(* PLC project measure36, PHOENIX CONTACT Software MULTIPROG 5.51 *)
(* stored: companyURL https://www.phoenixcontact-software.com, productRelease Build 473, creationDateTime 2024-06-25T14:51:15, contentDescription ###XMLINFO=2;1;2;;, version 0.1.75, modificationDateTime 2024-06-25T14:51:15 *)

PROGRAM mainST
  VAR
    input01 : BOOL;  (* 入力01 *)
    resLD : BOOL;
    resLDB : BOOL;
    C005 : BOOL;
    resAND : BOOL;
    C007 : BOOL;
    resANB : BOOL;
    C010 : BOOL;
    resOR : BOOL;
    C015 : BOOL;
    resORB : BOOL;
    resOUT : BOOL;
    resOUB : BOOL;
    resSET : BOOL;
    C024 : BOOL;
    resRES : BOOL;
    inTIMER01 : BOOL;
    TON_1 : TON;
    passed01 : TIME;
    TON_2 : TON;
    passed02 : TIME;
    resLD_T01 : BOOL;
    resLD_T02 : BOOL;
    inCounter : BOOL;
    enableCnt : BOOL;
    CTU_1 : CTU;
    outConter : BOOL;
    valCounter : INT;
    inTimER02 : BOOL;
    TON_3 : TON;
    passed03 : TIME;
    resT5 : BOOL;
    resLDB_T : BOOL;
    inCounter2 : BOOL;
    CTU_2 : CTU;
    outConter2 : BOOL;
    valCounter2 : INT;
    resLDB_C : BOOL;
    resLD_C : BOOL;
    inTimeR03 : BOOL;
    TON_4 : TON;
    outTimer : BOOL;
    passed04 : TIME;
    C046 : BOOL;
    resAND_T : BOOL;
    resTimer01 : BOOL;
    resTimer02 : BOOL;
    inCounter3 : BOOL;
    CTU_3 : CTU;
    outCounter3 : BOOL;
    valCounter3 : INT;
    C052 : BOOL;
    resAND_C : BOOL;
    inTimer05 : BOOL;
    TON_5 : TON;
    outTimer05 : BOOL;
    passed05 : TIME;
    C055 : BOOL;
    resANB_T : BOOL;
    inCounter04 : BOOL;
    CTU_4 : CTU;
    valCounter04 : INT;
    outConter04 : BOOL;
    C061 : BOOL;
    resANB_C : BOOL;
    inTimer06 : BOOL;
    TON_6 : TON;
    outTimer06 : BOOL;
    passed06 : TIME;
    resOR_T : BOOL;
    inCounter05 : BOOL;
    CTU_5 : CTU;
    outCounter05 : BOOL;
    valCounter05 : INT;
    resOR_C : BOOL;
    inTimer07 : BOOL;
    TON_7 : TON;
    outTimer07 : BOOL;
    passed07 : TIME;
    resORB_T : BOOL;
    inCounter06 : BOOL;
    CTU_6 : CTU;
    outCounter06 : BOOL;
    valCounter06 : INT;
    resORB_C : BOOL;
    C083 : BOOL;
    C085 : BOOL;
    resANL : BOOL;
    C089 : BOOL;
    C091 : BOOL;
    resORL : BOOL;
    setten0101 : BOOL;
    setten0102 : BOOL;
    setten0103 : BOOL;
    setten0104 : BOOL;
    resCoil01 : BOOL;
    setten0204 : BOOL;
    setten0304 : BOOL;
    resCoil02 : BOOL;
    resCoil03 : BOOL;
    setten0403 : BOOL;
    setten0503 : BOOL;
    resCoil04 : BOOL;
    resCoil05 : BOOL;
    setten0603 : BOOL;
    setten0702 : BOOL;
    setten0802 : BOOL;
    setten0902 : BOOL;
    resCoil07 : BOOL;
    resCoil06 : BOOL;
    resCoil08 : BOOL;
    resCoil09 : BOOL;
    C065 : BOOL;
    C069 : BOOL;
    C075 : BOOL;
    C078 : BOOL;
    inBia0101 : BOOL;
    inBia0102 : BOOL;
    inBia0202 : BOOL;
    inBia0203 : BOOL;
    inBia0303 : BOOL;
    inBIa0404 : BOOL;
    inBIa0504 : BOOL;
    resBia01 : BOOL;
    resBia02 : BOOL;
    resBia03 : BOOL;
    inCLR01 : BOOL;
    resCLR01 : BOOL;
    inCLR02 : BOOL;
    resCLR02 : BOOL;
    inCLR03 : BOOL;
    resCLR03 : BOOL;
    inCLR0401 : BOOL;
    inCLR0402 : BOOL;
    resCLR04 : BOOL;
    F_TRIG_1 : F_TRIG;
    inDIFU : BOOL;
    outDIFU : BOOL;
    resDIFU : BOOL;
    holdDIFU : BOOL;
    inDIFD : BOOL;
    R_TRIG_1 : R_TRIG;
    outDIFD : BOOL;
    holdDIFD : BOOL;
    resDIFD : BOOL;
    TotalCount : UINT;
    switch : BOOL;
  END_VAR
  VAR_EXTERNAL
    ECAT_Slave1_DI1 : BOOL;
  END_VAR
  VAR
    CTU_7 : CTU;
  END_VAR
  VAR_EXTERNAL
    ECAT_Slave4_AO1 : INT;
  END_VAR
  VAR
    CT_Reset : BOOL;
  END_VAR
  VAR_EXTERNAL
    ECAT_Slave5_DI1 : BOOL;
    ECAT_Slave5_DO1 : BOOL;
  END_VAR
  VAR
    IL変数_1 : BOOL;
    IL変数_2 : BOOL;
    IL変数_3 : BOOL;
    IL変数_4 : BOOL;
    IL変数_5 : BOOL;
    IL変数_6 : BOOL;
    IL変数_7 : BOOL;
    IL変数_8 : BOOL;
    IL変数_9 : BOOL;
    IL変数_10 : BOOL;
    IL変数_11 : BOOL;
    IL変数_12 : BOOL;
    IL変数_13 : BOOL;
    IL変数_14 : BOOL;
    IL変数_15 : BOOL;
    IL変数_16 : BOOL;
    IL変数_17 : BOOL;
    IL変数_18 : BOOL;
    IL変数_19 : BOOL;
    IL変数_20 : BOOL;
    IL変数_21 : BOOL;
    IL変数_22 : BOOL;
    IL変数_23 : BOOL;
    IL変数_24 : BOOL;
    IL変数_25 : BOOL;
    IL変数_26 : BOOL;
    IL変数_27 : BOOL;
    IL変数_28 : BOOL;
    IL変数_29 : BOOL;
    IL変数_30 : BOOL;
    IL変数_31 : BOOL;
    IL変数_32 : BOOL;
    IL変数_33 : BOOL;
    IL変数_34 : BOOL;
    IL変数_35 : BOOL;
    IL変数_36 : BOOL;
    IL変数_37 : BOOL;
    IL変数_38 : BOOL;
    IL変数_39 : BOOL;
    IL変数_40 : BOOL;
    IL変数_41 : BOOL;
    IL変数_42 : BOOL;
    IL変数_43 : BOOL;
    IL変数_44 : BOOL;
    IL変数_45 : BOOL;
    IL変数_46 : BOOL;
    IL変数_47 : BOOL;
    IL変数_48 : BOOL;
    IL変数_49 : BOOL;
    IL変数_50 : BOOL;
    IL変数_51 : BOOL;
    IL変数_52 : BOOL;
    IL変数_53 : BOOL;
    IL変数_54 : BOOL;
    IL変数_55 : BOOL;
    IL変数_56 : BOOL;
    IL変数_57 : BOOL;
    IL変数_58 : BOOL;
    IL変数_59 : BOOL;
    IL変数_60 : BOOL;
    IL変数_61 : BOOL;
    IL変数_62 : BOOL;
    IL変数_63 : BOOL;
    IL変数_64 : BOOL;
    IL変数_65 : BOOL;
    IL変数_66 : BOOL;
    IL変数_67 : BOOL;
    IL変数_68 : BOOL;
    IL変数_69 : BOOL;
    IL変数_70 : BOOL;
    IL変数_71 : BOOL;
    IL変数_72 : BOOL;
    IL変数_73 : BOOL;
    IL変数_74 : BOOL;
    IL変数_75 : BOOL;
    IL変数_76 : BOOL;
    IL変数_77 : BOOL;
    IL変数_78 : BOOL;
    IL変数_79 : BOOL;
    IL変数_80 : BOOL;
    IL変数_81 : BOOL;
    IL変数_82 : BOOL;
    IL変数_83 : BOOL;
    IL変数_84 : BOOL;
    IL変数_85 : BOOL;
    IL変数_86 : BOOL;
    IL変数_87 : BOOL;
    IL変数_88 : BOOL;
    IL変数_89 : BOOL;
    IL変数_90 : BOOL;
    IL変数_91 : BOOL;
    IL変数_92 : BOOL;
    IL変数_93 : BOOL;
    IL変数_94 : BOOL;
    IL変数_95 : BOOL;
    IL変数_96 : BOOL;
    IL変数_97 : BOOL;
    IL変数_98 : BOOL;
    IL変数_99 : BOOL;
    IL変数_100 : BOOL;
    IL変数_101 : BOOL;
    IL変数_102 : BOOL;
    IL変数_103 : BOOL;
    IL変数_104 : BOOL;
    IL変数_105 : BOOL;
    IL変数_106 : BOOL;
    IL変数_107 : BOOL;
    IL変数_108 : BOOL;
    IL変数_109 : BOOL;
    IL変数_110 : BOOL;
    IL変数_111 : BOOL;
    IL変数_112 : BOOL;
    IL変数_113 : BOOL;
    IL変数_114 : BOOL;
    IL変数_115 : BOOL;
    IL変数_116 : BOOL;
    IL変数_117 : BOOL;
    IL変数_118 : BOOL;
    IL変数_119 : BOOL;
    IL変数_120 : BOOL;
    IL変数_121 : BOOL;
    IL変数_122 : BOOL;
    IL変数_123 : BOOL;
    IL変数_124 : BOOL;
    IL変数_125 : BOOL;
    IL変数_126 : BOOL;
    IL変数_127 : BOOL;
    IL変数_128 : BOOL;
    IL変数_129 : BOOL;
    IL変数_130 : BOOL;
    IL変数_131 : BOOL;
    IL変数_132 : BOOL;
    IL変数_133 : BOOL;
    IL変数_134 : BOOL;
    IL変数_135 : BOOL;
    IL変数_136 : BOOL;
    IL変数_137 : BOOL;
    IL変数_138 : BOOL;
    IL変数_139 : BOOL;
    IL変数_140 : BOOL;
    IL変数_141 : BOOL;
    IL変数_142 : BOOL;
    IL変数_143 : BOOL;
    IL変数_144 : BOOL;
    IL変数_145 : BOOL;
    IL変数_146 : BOOL;
    IL変数_147 : BOOL;
    IL変数_148 : BOOL;
    IL変数_149 : BOOL;
    IL変数_150 : BOOL;
    IL変数_151 : BOOL;
    IL変数_152 : BOOL;
    IL変数_153 : BOOL;
    IL変数_154 : BOOL;
    IL変数_155 : BOOL;
    IL変数_156 : BOOL;
    IL変数_157 : BOOL;
    IL変数_158 : BOOL;
    IL変数_159 : BOOL;
    IL変数_160 : BOOL;
    IL変数_161 : BOOL;
    IL変数_162 : BOOL;
    IL変数_163 : BOOL;
    IL変数_164 : BOOL;
    IL変数_165 : BOOL;
    IL変数_166 : BOOL;
    IL変数_167 : BOOL;
    IL変数_168 : BOOL;
    IL変数_169 : BOOL;
    IL変数_170 : BOOL;
    IL変数_171 : BOOL;
    IL変数_172 : BOOL;
    IL変数_173 : BOOL;
    IL変数_174 : BOOL;
    IL変数_175 : BOOL;
    IL変数_176 : BOOL;
    IL変数_177 : BOOL;
    IL変数_178 : BOOL;
    IL変数_179 : BOOL;
    IL変数_180 : BOOL;
  END_VAR

						
							
								
							
							
								(**** 全命令テスト ****)
(**** 回路ON ****)
LD		ECAT_Slave5_DI1
ST		input01
ST		inBia0101
ST		inBia0102
ST		inBia0202
ST		inBia0203
ST		inBia0303
ST		inBIa0404
ST		inBIa0504
ST		inCLR01
ST		inCLR02
ST		inCLR03
ST		inCLR0401
ST		inCLR0402
ST		inCounter
ST		inCounter2
ST		inCounter3
ST		inCounter04
ST		inCounter05
ST		inCounter06
ST		inDIFU
ST		inDIFD
ST		inTIMER01
ST		inTimER02
ST		inTimeR03
ST		inTimer05
ST		inTimer06
ST		inTimer07
									
								
							
						
					
						
							
								
							
							
								(*■LD命令*)
LD		input01
ST		resLD
									
(*■LDB命令*)
LDN		input01
STN		resLDB
									
(*■AND命令*)
LDN		C005
AND		input01
ST		resAND
									
(*■ANB命令*)
LDN		C007
ANDN		input01
STN		resANB
									
(*■OR命令*)
LD		C010
OR		input01
ST		resOR
									
(*■ORB命令*)
LD		C015
ORN		input01
STN		resORB
									
(*■OUT命令*)
LD		input01
ST		resOUT
									
(*■OUB命令*)
LDN		input01
STN		resOUB
									
(*■SET命令*)
LD		input01
ANDN		resSET
S		resSET
									
(*■RES命令*)
LD		input01
S		C024
									
LD		input01
R		C024
									
LDN		C024
ST		resRES
									
(*■LD_T命令*)
LD		inTIMER01
ST		TON_1.IN
ST		TON_2.IN
LD		TIME#30s
ST		TON_1.PT
CAL		TON_1
LD		TON_1.Q
ST		resTimer01
LD		TON_1.ET
ST		passed01
LD		TIME#1m
ST		TON_2.PT
CAL		TON_2
LD		TON_2.Q
ST		resTimer02
LD		TON_2.ET
ST		passed02
									
LD		resTimer01
ST		resLD_T01
									
LD		resTimer02
ST		resLD_T02
									
(*■LD_C命令*)
LD		inCounter
ST		CTU_1.CU
LD		enableCnt
ST		CTU_1.RESET
LD		INT#5000
ST		CTU_1.PV
CAL		CTU_1
LD		CTU_1.Q
ST		outConter
LD		CTU_1.CV
ST		valCounter
									
LD		outConter
ST		resLD_C
									
(*■LDB_T命令*)
LD		inTimER02
ST		TON_3.IN
LD		TIME#30s
ST		TON_3.PT
CAL		TON_3
LD		TON_3.Q
ST		resT5
LD		TON_3.ET
ST		passed03
									
LDN		resT5
STN		resLDB_T
									
(*■LDB_C命令*)
LD		inCounter2
ST		CTU_2.CU
LD		enableCnt
ST		CTU_2.RESET
LD		INT#5000
ST		CTU_2.PV
CAL		CTU_2
LD		CTU_2.Q
ST		outConter2
LD		CTU_2.CV
ST		valCounter2
									
LDN		outConter2
STN		resLDB_C
									
(*■AND_T命令*)
LD		inTimeR03
ST		TON_4.IN
LD		TIME#30s
ST		TON_4.PT
CAL		TON_4
LD		TON_4.Q
ST		outTimer
LD		TON_4.ET
ST		passed04
									
LDN		C046
AND		outTimer
ST		resAND_T
									
(*■AND_C命令*)
LD		inCounter3
ST		CTU_3.CU
LD		enableCnt
ST		CTU_3.RESET
LD		INT#5000
ST		CTU_3.PV
CAL		CTU_3
LD		CTU_3.Q
ST		outCounter3
LD		CTU_3.CV
ST		valCounter3
									
LDN		C052
AND		outCounter3
ST		resAND_C
									
(*■ANB_T命令*)
LD		inTimer05
ST		TON_5.IN
LD		TIME#30s
ST		TON_5.PT
CAL		TON_5
LD		TON_5.Q
ST		outTimer05
LD		TON_5.ET
ST		passed05
									
LDN		C055
ANDN		outTimer05
STN		resANB_T
									
(*■ANB_C命令*)
LD		inCounter04
ST		CTU_4.CU
LD		enableCnt
ST		CTU_4.RESET
LD		INT#5000
ST		CTU_4.PV
CAL		CTU_4
LD		CTU_4.Q
ST		outConter04
LD		CTU_4.CV
ST		valCounter04
									
LDN		C061
ANDN		outConter04
STN		resANB_C
									
(*■OR_T命令*)
LD		inTimer06
ST		TON_6.IN
LD		TIME#30s
ST		TON_6.PT
CAL		TON_6
LD		TON_6.Q
ST		outTimer06
LD		TON_6.ET
ST		passed06
									
LD		C065
OR		outTimer06
ST		resOR_T
									
(*■OR_C命令*)
LD		inCounter05
ST		CTU_5.CU
LD		enableCnt
ST		CTU_5.RESET
LD		INT#5000
ST		CTU_5.PV
CAL		CTU_5
LD		CTU_5.Q
ST		outCounter05
LD		CTU_5.CV
ST		valCounter05
									
LD		C069
OR		outCounter05
ST		resOR_C
									
(*■ORB_T命令*)
LD		inTimer07
ST		TON_7.IN
LD		TIME#30s
ST		TON_7.PT
CAL		TON_7
LD		TON_7.Q
ST		outTimer07
LD		TON_7.ET
ST		passed07
									
LD		C075
ORN		outTimer07
STN		resORB_T
									
(*■ORB_C命令*)
LD		inCounter06
ST		CTU_6.CU
LD		enableCnt
ST		CTU_6.RESET
LD		INT#5000
ST		CTU_6.PV
CAL		CTU_6
LD		CTU_6.Q
ST		outCounter06
LD		CTU_6.CV
ST		valCounter06
									
LD		C078
ORN		outCounter06
STN		resORB_C
									
(*■ANL命令*)
LD		input01
OR		C083
ST		IL変数_1
LD		input01
OR		C085
AND		IL変数_1
ST		resANL
									
(*■ORL命令*)
LD		input01
AND		input01
ST		IL変数_2
LD		C089
AND		C091
OR		IL変数_2
ST		resORL
									
(*■MPS、MPP、MRD命令*)
LD		setten0101
AND		setten0102
ST		IL変数_3
LD		IL変数_3
AND		setten0103
ST		IL変数_4
LD		IL変数_4
AND		setten0104
ST		resCoil01
LD		IL変数_4
AND		setten0204
ST		resCoil02
LD		IL変数_4
AND		setten0304
ST		resCoil03
LD		IL変数_3
AND		setten0403
ST		resCoil04
LD		IL変数_3
AND		setten0503
ST		resCoil05
LD		IL変数_3
AND		setten0603
ST		resCoil06
									
LD		setten0101
AND		setten0702
ST		resCoil07
									
LD		setten0101
AND		setten0802
ST		resCoil08
									
LD		setten0101
AND		setten0902
ST		resCoil09
									
(*■ビアメカ問題発生ロジック*)
LD		inBia0102
OR		inBia0202
AND		inBia0101
ST		resBia01
LD		resBia01
AND		inBia0203
ST		resBia02
LD		inBIa0404
OR		inBIa0504
ST		IL変数_5
LD		resBia01
AND		inBia0303
AND		IL変数_5
ST		resBia03
									
(*■CLR命令*)
(*実行されるパターン*)
LD		inCLR01
ST		resCLR01
									
LD		inCLR02
ST		resCLR02
									
(*実行されないパターン*)
LD		inCLR03
ST		resCLR03
AND		inCLR0401
AND		inCLR0402
ST		resCLR04
									
(*■DIFU(TRIGON)命令*)
LD		inDIFU
ST		R_TRIG_1.CLK
CAL		R_TRIG_1
LD		R_TRIG_1.Q
ST		outDIFU
									
LD		outDIFU
OR		holdDIFU
ST		holdDIFU
									
LDN		outDIFU
AND		holdDIFU
ST		resDIFU
									
(*■DIFD(TRIGOFF)命令*)
LD		inDIFD
ST		F_TRIG_1.CLK
CAL		F_TRIG_1
LD		F_TRIG_1.Q
ST		outDIFD
									
LD		outDIFD
OR		holdDIFD
ST		holdDIFD
									
(*-----ここまで-----------------------------------------------------
*)
LD		holdDIFD
ANDN		outDIFD
ST		resDIFD
									
								
							
						
					
						
							
								
							
							
								(*■LD命令*)
LD		input01
ST		resLD
									
(*■LDB命令*)
LDN		input01
STN		resLDB
									
(*■AND命令*)
LDN		C005
AND		input01
ST		resAND
									
(*■ANB命令*)
LDN		C007
ANDN		input01
STN		resANB
									
(*■OR命令*)
LD		C010
OR		input01
ST		resOR
									
(*■ORB命令*)
LD		C015
ORN		input01
STN		resORB
									
(*■OUT命令*)
LD		input01
ST		resOUT
									
(*■OUB命令*)
LDN		input01
STN		resOUB
									
(*■SET命令*)
LD		input01
ANDN		resSET
S		resSET
									
(*■RES命令*)
LD		input01
S		C024
									
LD		input01
R		C024
									
LDN		C024
ST		resRES
									
(*■LD_T命令*)
LD		inTIMER01
ST		TON_1.IN
ST		TON_2.IN
LD		TIME#30s
ST		TON_1.PT
CAL		TON_1
LD		TON_1.Q
ST		resTimer01
LD		TON_1.ET
ST		passed01
LD		TIME#1m
ST		TON_2.PT
CAL		TON_2
LD		TON_2.Q
ST		resTimer02
LD		TON_2.ET
ST		passed02
									
LD		resTimer01
ST		resLD_T01
									
LD		resTimer02
ST		resLD_T02
									
(*■LD_C命令*)
LD		inCounter
ST		CTU_1.CU
LD		enableCnt
ST		CTU_1.RESET
LD		INT#5000
ST		CTU_1.PV
CAL		CTU_1
LD		CTU_1.Q
ST		outConter
LD		CTU_1.CV
ST		valCounter
									
LD		outConter
ST		resLD_C
									
(*■LDB_T命令*)
LD		inTimER02
ST		TON_3.IN
LD		TIME#30s
ST		TON_3.PT
CAL		TON_3
LD		TON_3.Q
ST		resT5
LD		TON_3.ET
ST		passed03
									
LDN		resT5
STN		resLDB_T
									
(*■LDB_C命令*)
LD		inCounter2
ST		CTU_2.CU
LD		enableCnt
ST		CTU_2.RESET
LD		INT#5000
ST		CTU_2.PV
CAL		CTU_2
LD		CTU_2.Q
ST		outConter2
LD		CTU_2.CV
ST		valCounter2
									
LDN		outConter2
STN		resLDB_C
									
(*■AND_T命令*)
LD		inTimeR03
ST		TON_4.IN
LD		TIME#30s
ST		TON_4.PT
CAL		TON_4
LD		TON_4.Q
ST		outTimer
LD		TON_4.ET
ST		passed04
									
LDN		C046
AND		outTimer
ST		resAND_T
									
(*■AND_C命令*)
LD		inCounter3
ST		CTU_3.CU
LD		enableCnt
ST		CTU_3.RESET
LD		INT#5000
ST		CTU_3.PV
CAL		CTU_3
LD		CTU_3.Q
ST		outCounter3
LD		CTU_3.CV
ST		valCounter3
									
LDN		C052
AND		outCounter3
ST		resAND_C
									
(*■ANB_T命令*)
LD		inTimer05
ST		TON_5.IN
LD		TIME#30s
ST		TON_5.PT
CAL		TON_5
LD		TON_5.Q
ST		outTimer05
LD		TON_5.ET
ST		passed05
									
LDN		C055
ANDN		outTimer05
STN		resANB_T
									
(*■ANB_C命令*)
LD		inCounter04
ST		CTU_4.CU
LD		enableCnt
ST		CTU_4.RESET
LD		INT#5000
ST		CTU_4.PV
CAL		CTU_4
LD		CTU_4.Q
ST		outConter04
LD		CTU_4.CV
ST		valCounter04
									
LDN		C061
ANDN		outConter04
STN		resANB_C
									
(*■OR_T命令*)
LD		inTimer06
ST		TON_6.IN
LD		TIME#30s
ST		TON_6.PT
CAL		TON_6
LD		TON_6.Q
ST		outTimer06
LD		TON_6.ET
ST		passed06
									
LD		C065
OR		outTimer06
ST		resOR_T
									
(*■OR_C命令*)
LD		inCounter05
ST		CTU_5.CU
LD		enableCnt
ST		CTU_5.RESET
LD		INT#5000
ST		CTU_5.PV
CAL		CTU_5
LD		CTU_5.Q
ST		outCounter05
LD		CTU_5.CV
ST		valCounter05
									
LD		C069
OR		outCounter05
ST		resOR_C
									
(*■ORB_T命令*)
LD		inTimer07
ST		TON_7.IN
LD		TIME#30s
ST		TON_7.PT
CAL		TON_7
LD		TON_7.Q
ST		outTimer07
LD		TON_7.ET
ST		passed07
									
LD		C075
ORN		outTimer07
STN		resORB_T
									
(*■ORB_C命令*)
LD		inCounter06
ST		CTU_6.CU
LD		enableCnt
ST		CTU_6.RESET
LD		INT#5000
ST		CTU_6.PV
CAL		CTU_6
LD		CTU_6.Q
ST		outCounter06
LD		CTU_6.CV
ST		valCounter06
									
LD		C078
ORN		outCounter06
STN		resORB_C
									
(*■ANL命令*)
LD		input01
OR		C083
ST		IL変数_6
LD		input01
OR		C085
AND		IL変数_6
ST		resANL
									
(*■ORL命令*)
LD		input01
AND		input01
ST		IL変数_7
LD		C089
AND		C091
OR		IL変数_7
ST		resORL
									
(*■MPS、MPP、MRD命令*)
LD		setten0101
AND		setten0102
ST		IL変数_8
LD		IL変数_8
AND		setten0103
ST		IL変数_9
LD		IL変数_9
AND		setten0104
ST		resCoil01
LD		IL変数_9
AND		setten0204
ST		resCoil02
LD		IL変数_9
AND		setten0304
ST		resCoil03
LD		IL変数_8
AND		setten0403
ST		resCoil04
LD		IL変数_8
AND		setten0503
ST		resCoil05
LD		IL変数_8
AND		setten0603
ST		resCoil06
									
LD		setten0101
AND		setten0702
ST		resCoil07
									
LD		setten0101
AND		setten0802
ST		resCoil08
									
LD		setten0101
AND		setten0902
ST		resCoil09
									
(*■ビアメカ問題発生ロジック*)
LD		inBia0102
OR		inBia0202
AND		inBia0101
ST		resBia01
LD		resBia01
AND		inBia0203
ST		resBia02
LD		inBIa0404
OR		inBIa0504
ST		IL変数_10
LD		resBia01
AND		inBia0303
AND		IL変数_10
ST		resBia03
									
(*■CLR命令*)
(*実行されるパターン*)
LD		inCLR01
ST		resCLR01
									
LD		inCLR02
ST		resCLR02
									
(*実行されないパターン*)
LD		inCLR03
ST		resCLR03
AND		inCLR0401
AND		inCLR0402
ST		resCLR04
									
(*■DIFU(TRIGON)命令*)
LD		inDIFU
ST		R_TRIG_1.CLK
CAL		R_TRIG_1
LD		R_TRIG_1.Q
ST		outDIFU
									
LD		outDIFU
OR		holdDIFU
ST		holdDIFU
									
LDN		outDIFU
AND		holdDIFU
ST		resDIFU
									
(*■DIFD(TRIGOFF)命令*)
LD		inDIFD
ST		F_TRIG_1.CLK
CAL		F_TRIG_1
LD		F_TRIG_1.Q
ST		outDIFD
									
LD		outDIFD
OR		holdDIFD
ST		holdDIFD
									
(*-----ここまで-----------------------------------------------------
*)
LD		holdDIFD
ANDN		outDIFD
ST		resDIFD
									
								
							
						
					
						
							
								
							
							
								(*■LD命令*)
LD		input01
ST		resLD
									
(*■LDB命令*)
LDN		input01
STN		resLDB
									
(*■AND命令*)
LDN		C005
AND		input01
ST		resAND
									
(*■ANB命令*)
LDN		C007
ANDN		input01
STN		resANB
									
(*■OR命令*)
LD		C010
OR		input01
ST		resOR
									
(*■ORB命令*)
LD		C015
ORN		input01
STN		resORB
									
(*■OUT命令*)
LD		input01
ST		resOUT
									
(*■OUB命令*)
LDN		input01
STN		resOUB
									
(*■SET命令*)
LD		input01
ANDN		resSET
S		resSET
									
(*■RES命令*)
LD		input01
S		C024
									
LD		input01
R		C024
									
LDN		C024
ST		resRES
									
(*■LD_T命令*)
LD		inTIMER01
ST		TON_1.IN
ST		TON_2.IN
LD		TIME#30s
ST		TON_1.PT
CAL		TON_1
LD		TON_1.Q
ST		resTimer01
LD		TON_1.ET
ST		passed01
LD		TIME#1m
ST		TON_2.PT
CAL		TON_2
LD		TON_2.Q
ST		resTimer02
LD		TON_2.ET
ST		passed02
									
LD		resTimer01
ST		resLD_T01
									
LD		resTimer02
ST		resLD_T02
									
(*■LD_C命令*)
LD		inCounter
ST		CTU_1.CU
LD		enableCnt
ST		CTU_1.RESET
LD		INT#5000
ST		CTU_1.PV
CAL		CTU_1
LD		CTU_1.Q
ST		outConter
LD		CTU_1.CV
ST		valCounter
									
LD		outConter
ST		resLD_C
									
(*■LDB_T命令*)
LD		inTimER02
ST		TON_3.IN
LD		TIME#30s
ST		TON_3.PT
CAL		TON_3
LD		TON_3.Q
ST		resT5
LD		TON_3.ET
ST		passed03
									
LDN		resT5
STN		resLDB_T
									
(*■LDB_C命令*)
LD		inCounter2
ST		CTU_2.CU
LD		enableCnt
ST		CTU_2.RESET
LD		INT#5000
ST		CTU_2.PV
CAL		CTU_2
LD		CTU_2.Q
ST		outConter2
LD		CTU_2.CV
ST		valCounter2
									
LDN		outConter2
STN		resLDB_C
									
(*■AND_T命令*)
LD		inTimeR03
ST		TON_4.IN
LD		TIME#30s
ST		TON_4.PT
CAL		TON_4
LD		TON_4.Q
ST		outTimer
LD		TON_4.ET
ST		passed04
									
LDN		C046
AND		outTimer
ST		resAND_T
									
(*■AND_C命令*)
LD		inCounter3
ST		CTU_3.CU
LD		enableCnt
ST		CTU_3.RESET
LD		INT#5000
ST		CTU_3.PV
CAL		CTU_3
LD		CTU_3.Q
ST		outCounter3
LD		CTU_3.CV
ST		valCounter3
									
LDN		C052
AND		outCounter3
ST		resAND_C
									
(*■ANB_T命令*)
LD		inTimer05
ST		TON_5.IN
LD		TIME#30s
ST		TON_5.PT
CAL		TON_5
LD		TON_5.Q
ST		outTimer05
LD		TON_5.ET
ST		passed05
									
LDN		C055
ANDN		outTimer05
STN		resANB_T
									
(*■ANB_C命令*)
LD		inCounter04
ST		CTU_4.CU
LD		enableCnt
ST		CTU_4.RESET
LD		INT#5000
ST		CTU_4.PV
CAL		CTU_4
LD		CTU_4.Q
ST		outConter04
LD		CTU_4.CV
ST		valCounter04
									
LDN		C061
ANDN		outConter04
STN		resANB_C
									
(*■OR_T命令*)
LD		inTimer06
ST		TON_6.IN
LD		TIME#30s
ST		TON_6.PT
CAL		TON_6
LD		TON_6.Q
ST		outTimer06
LD		TON_6.ET
ST		passed06
									
LD		C065
OR		outTimer06
ST		resOR_T
									
(*■OR_C命令*)
LD		inCounter05
ST		CTU_5.CU
LD		enableCnt
ST		CTU_5.RESET
LD		INT#5000
ST		CTU_5.PV
CAL		CTU_5
LD		CTU_5.Q
ST		outCounter05
LD		CTU_5.CV
ST		valCounter05
									
LD		C069
OR		outCounter05
ST		resOR_C
									
(*■ORB_T命令*)
LD		inTimer07
ST		TON_7.IN
LD		TIME#30s
ST		TON_7.PT
CAL		TON_7
LD		TON_7.Q
ST		outTimer07
LD		TON_7.ET
ST		passed07
									
LD		C075
ORN		outTimer07
STN		resORB_T
									
(*■ORB_C命令*)
LD		inCounter06
ST		CTU_6.CU
LD		enableCnt
ST		CTU_6.RESET
LD		INT#5000
ST		CTU_6.PV
CAL		CTU_6
LD		CTU_6.Q
ST		outCounter06
LD		CTU_6.CV
ST		valCounter06
									
LD		C078
ORN		outCounter06
STN		resORB_C
									
(*■ANL命令*)
LD		input01
OR		C083
ST		IL変数_11
LD		input01
OR		C085
AND		IL変数_11
ST		resANL
									
(*■ORL命令*)
LD		input01
AND		input01
ST		IL変数_12
LD		C089
AND		C091
OR		IL変数_12
ST		resORL
									
(*■MPS、MPP、MRD命令*)
LD		setten0101
AND		setten0102
ST		IL変数_13
LD		IL変数_13
AND		setten0103
ST		IL変数_14
LD		IL変数_14
AND		setten0104
ST		resCoil01
LD		IL変数_14
AND		setten0204
ST		resCoil02
LD		IL変数_14
AND		setten0304
ST		resCoil03
LD		IL変数_13
AND		setten0403
ST		resCoil04
LD		IL変数_13
AND		setten0503
ST		resCoil05
LD		IL変数_13
AND		setten0603
ST		resCoil06
									
LD		setten0101
AND		setten0702
ST		resCoil07
									
LD		setten0101
AND		setten0802
ST		resCoil08
									
LD		setten0101
AND		setten0902
ST		resCoil09
									
(*■ビアメカ問題発生ロジック*)
LD		inBia0102
OR		inBia0202
AND		inBia0101
ST		resBia01
LD		resBia01
AND		inBia0203
ST		resBia02
LD		inBIa0404
OR		inBIa0504
ST		IL変数_15
LD		resBia01
AND		inBia0303
AND		IL変数_15
ST		resBia03
									
(*■CLR命令*)
(*実行されるパターン*)
LD		inCLR01
ST		resCLR01
									
LD		inCLR02
ST		resCLR02
									
(*実行されないパターン*)
LD		inCLR03
ST		resCLR03
AND		inCLR0401
AND		inCLR0402
ST		resCLR04
									
(*■DIFU(TRIGON)命令*)
LD		inDIFU
ST		R_TRIG_1.CLK
CAL		R_TRIG_1
LD		R_TRIG_1.Q
ST		outDIFU
									
LD		outDIFU
OR		holdDIFU
ST		holdDIFU
									
LDN		outDIFU
AND		holdDIFU
ST		resDIFU
									
(*■DIFD(TRIGOFF)命令*)
LD		inDIFD
ST		F_TRIG_1.CLK
CAL		F_TRIG_1
LD		F_TRIG_1.Q
ST		outDIFD
									
LD		outDIFD
OR		holdDIFD
ST		holdDIFD
									
(*-----ここまで-----------------------------------------------------
*)
LD		holdDIFD
ANDN		outDIFD
ST		resDIFD
									
								
							
						
					
						
							
								
							
							
								(*■LD命令*)
LD		input01
ST		resLD
									
(*■LDB命令*)
LDN		input01
STN		resLDB
									
(*■AND命令*)
LDN		C005
AND		input01
ST		resAND
									
(*■ANB命令*)
LDN		C007
ANDN		input01
STN		resANB
									
(*■OR命令*)
LD		C010
OR		input01
ST		resOR
									
(*■ORB命令*)
LD		C015
ORN		input01
STN		resORB
									
(*■OUT命令*)
LD		input01
ST		resOUT
									
(*■OUB命令*)
LDN		input01
STN		resOUB
									
(*■SET命令*)
LD		input01
ANDN		resSET
S		resSET
									
(*■RES命令*)
LD		input01
S		C024
									
LD		input01
R		C024
									
LDN		C024
ST		resRES
									
(*■LD_T命令*)
LD		inTIMER01
ST		TON_1.IN
ST		TON_2.IN
LD		TIME#30s
ST		TON_1.PT
CAL		TON_1
LD		TON_1.Q
ST		resTimer01
LD		TON_1.ET
ST		passed01
LD		TIME#1m
ST		TON_2.PT
CAL		TON_2
LD		TON_2.Q
ST		resTimer02
LD		TON_2.ET
ST		passed02
									
LD		resTimer01
ST		resLD_T01
									
LD		resTimer02
ST		resLD_T02
									
(*■LD_C命令*)
LD		inCounter
ST		CTU_1.CU
LD		enableCnt
ST		CTU_1.RESET
LD		INT#5000
ST		CTU_1.PV
CAL		CTU_1
LD		CTU_1.Q
ST		outConter
LD		CTU_1.CV
ST		valCounter
									
LD		outConter
ST		resLD_C
									
(*■LDB_T命令*)
LD		inTimER02
ST		TON_3.IN
LD		TIME#30s
ST		TON_3.PT
CAL		TON_3
LD		TON_3.Q
ST		resT5
LD		TON_3.ET
ST		passed03
									
LDN		resT5
STN		resLDB_T
									
(*■LDB_C命令*)
LD		inCounter2
ST		CTU_2.CU
LD		enableCnt
ST		CTU_2.RESET
LD		INT#5000
ST		CTU_2.PV
CAL		CTU_2
LD		CTU_2.Q
ST		outConter2
LD		CTU_2.CV
ST		valCounter2
									
LDN		outConter2
STN		resLDB_C
									
(*■AND_T命令*)
LD		inTimeR03
ST		TON_4.IN
LD		TIME#30s
ST		TON_4.PT
CAL		TON_4
LD		TON_4.Q
ST		outTimer
LD		TON_4.ET
ST		passed04
									
LDN		C046
AND		outTimer
ST		resAND_T
									
(*■AND_C命令*)
LD		inCounter3
ST		CTU_3.CU
LD		enableCnt
ST		CTU_3.RESET
LD		INT#5000
ST		CTU_3.PV
CAL		CTU_3
LD		CTU_3.Q
ST		outCounter3
LD		CTU_3.CV
ST		valCounter3
									
LDN		C052
AND		outCounter3
ST		resAND_C
									
(*■ANB_T命令*)
LD		inTimer05
ST		TON_5.IN
LD		TIME#30s
ST		TON_5.PT
CAL		TON_5
LD		TON_5.Q
ST		outTimer05
LD		TON_5.ET
ST		passed05
									
LDN		C055
ANDN		outTimer05
STN		resANB_T
									
(*■ANB_C命令*)
LD		inCounter04
ST		CTU_4.CU
LD		enableCnt
ST		CTU_4.RESET
LD		INT#5000
ST		CTU_4.PV
CAL		CTU_4
LD		CTU_4.Q
ST		outConter04
LD		CTU_4.CV
ST		valCounter04
									
LDN		C061
ANDN		outConter04
STN		resANB_C
									
(*■OR_T命令*)
LD		inTimer06
ST		TON_6.IN
LD		TIME#30s
ST		TON_6.PT
CAL		TON_6
LD		TON_6.Q
ST		outTimer06
LD		TON_6.ET
ST		passed06
									
LD		C065
OR		outTimer06
ST		resOR_T
									
(*■OR_C命令*)
LD		inCounter05
ST		CTU_5.CU
LD		enableCnt
ST		CTU_5.RESET
LD		INT#5000
ST		CTU_5.PV
CAL		CTU_5
LD		CTU_5.Q
ST		outCounter05
LD		CTU_5.CV
ST		valCounter05
									
LD		C069
OR		outCounter05
ST		resOR_C
									
(*■ORB_T命令*)
LD		inTimer07
ST		TON_7.IN
LD		TIME#30s
ST		TON_7.PT
CAL		TON_7
LD		TON_7.Q
ST		outTimer07
LD		TON_7.ET
ST		passed07
									
LD		C075
ORN		outTimer07
STN		resORB_T
									
(*■ORB_C命令*)
LD		inCounter06
ST		CTU_6.CU
LD		enableCnt
ST		CTU_6.RESET
LD		INT#5000
ST		CTU_6.PV
CAL		CTU_6
LD		CTU_6.Q
ST		outCounter06
LD		CTU_6.CV
ST		valCounter06
									
LD		C078
ORN		outCounter06
STN		resORB_C
									
(*■ANL命令*)
LD		input01
OR		C083
ST		IL変数_16
LD		input01
OR		C085
AND		IL変数_16
ST		resANL
									
(*■ORL命令*)
LD		input01
AND		input01
ST		IL変数_17
LD		C089
AND		C091
OR		IL変数_17
ST		resORL
									
(*■MPS、MPP、MRD命令*)
LD		setten0101
AND		setten0102
ST		IL変数_18
LD		IL変数_18
AND		setten0103
ST		IL変数_19
LD		IL変数_19
AND		setten0104
ST		resCoil01
LD		IL変数_19
AND		setten0204
ST		resCoil02
LD		IL変数_19
AND		setten0304
ST		resCoil03
LD		IL変数_18
AND		setten0403
ST		resCoil04
LD		IL変数_18
AND		setten0503
ST		resCoil05
LD		IL変数_18
AND		setten0603
ST		resCoil06
									
LD		setten0101
AND		setten0702
ST		resCoil07
									
LD		setten0101
AND		setten0802
ST		resCoil08
									
LD		setten0101
AND		setten0902
ST		resCoil09
									
(*■ビアメカ問題発生ロジック*)
LD		inBia0102
OR		inBia0202
AND		inBia0101
ST		resBia01
LD		resBia01
AND		inBia0203
ST		resBia02
LD		inBIa0404
OR		inBIa0504
ST		IL変数_20
LD		resBia01
AND		inBia0303
AND		IL変数_20
ST		resBia03
									
(*■CLR命令*)
(*実行されるパターン*)
LD		inCLR01
ST		resCLR01
									
LD		inCLR02
ST		resCLR02
									
(*実行されないパターン*)
LD		inCLR03
ST		resCLR03
AND		inCLR0401
AND		inCLR0402
ST		resCLR04
									
(*■DIFU(TRIGON)命令*)
LD		inDIFU
ST		R_TRIG_1.CLK
CAL		R_TRIG_1
LD		R_TRIG_1.Q
ST		outDIFU
									
LD		outDIFU
OR		holdDIFU
ST		holdDIFU
									
LDN		outDIFU
AND		holdDIFU
ST		resDIFU
									
(*■DIFD(TRIGOFF)命令*)
LD		inDIFD
ST		F_TRIG_1.CLK
CAL		F_TRIG_1
LD		F_TRIG_1.Q
ST		outDIFD
									
LD		outDIFD
OR		holdDIFD
ST		holdDIFD
									
(*-----ここまで-----------------------------------------------------
*)
LD		holdDIFD
ANDN		outDIFD
ST		resDIFD
									
								
							
						
					
						
							
								
							
							
								(*■LD命令*)
LD		input01
ST		resLD
									
(*■LDB命令*)
LDN		input01
STN		resLDB
									
(*■AND命令*)
LDN		C005
AND		input01
ST		resAND
									
(*■ANB命令*)
LDN		C007
ANDN		input01
STN		resANB
									
(*■OR命令*)
LD		C010
OR		input01
ST		resOR
									
(*■ORB命令*)
LD		C015
ORN		input01
STN		resORB
									
(*■OUT命令*)
LD		input01
ST		resOUT
									
(*■OUB命令*)
LDN		input01
STN		resOUB
									
(*■SET命令*)
LD		input01
ANDN		resSET
S		resSET
									
(*■RES命令*)
LD		input01
S		C024
									
LD		input01
R		C024
									
LDN		C024
ST		resRES
									
(*■LD_T命令*)
LD		inTIMER01
ST		TON_1.IN
ST		TON_2.IN
LD		TIME#30s
ST		TON_1.PT
CAL		TON_1
LD		TON_1.Q
ST		resTimer01
LD		TON_1.ET
ST		passed01
LD		TIME#1m
ST		TON_2.PT
CAL		TON_2
LD		TON_2.Q
ST		resTimer02
LD		TON_2.ET
ST		passed02
									
LD		resTimer01
ST		resLD_T01
									
LD		resTimer02
ST		resLD_T02
									
(*■LD_C命令*)
LD		inCounter
ST		CTU_1.CU
LD		enableCnt
ST		CTU_1.RESET
LD		INT#5000
ST		CTU_1.PV
CAL		CTU_1
LD		CTU_1.Q
ST		outConter
LD		CTU_1.CV
ST		valCounter
									
LD		outConter
ST		resLD_C
									
(*■LDB_T命令*)
LD		inTimER02
ST		TON_3.IN
LD		TIME#30s
ST		TON_3.PT
CAL		TON_3
LD		TON_3.Q
ST		resT5
LD		TON_3.ET
ST		passed03
									
LDN		resT5
STN		resLDB_T
									
(*■LDB_C命令*)
LD		inCounter2
ST		CTU_2.CU
LD		enableCnt
ST		CTU_2.RESET
LD		INT#5000
ST		CTU_2.PV
CAL		CTU_2
LD		CTU_2.Q
ST		outConter2
LD		CTU_2.CV
ST		valCounter2
									
LDN		outConter2
STN		resLDB_C
									
(*■AND_T命令*)
LD		inTimeR03
ST		TON_4.IN
LD		TIME#30s
ST		TON_4.PT
CAL		TON_4
LD		TON_4.Q
ST		outTimer
LD		TON_4.ET
ST		passed04
									
LDN		C046
AND		outTimer
ST		resAND_T
									
(*■AND_C命令*)
LD		inCounter3
ST		CTU_3.CU
LD		enableCnt
ST		CTU_3.RESET
LD		INT#5000
ST		CTU_3.PV
CAL		CTU_3
LD		CTU_3.Q
ST		outCounter3
LD		CTU_3.CV
ST		valCounter3
									
LDN		C052
AND		outCounter3
ST		resAND_C
									
(*■ANB_T命令*)
LD		inTimer05
ST		TON_5.IN
LD		TIME#30s
ST		TON_5.PT
CAL		TON_5
LD		TON_5.Q
ST		outTimer05
LD		TON_5.ET
ST		passed05
									
LDN		C055
ANDN		outTimer05
STN		resANB_T
									
(*■ANB_C命令*)
LD		inCounter04
ST		CTU_4.CU
LD		enableCnt
ST		CTU_4.RESET
LD		INT#5000
ST		CTU_4.PV
CAL		CTU_4
LD		CTU_4.Q
ST		outConter04
LD		CTU_4.CV
ST		valCounter04
									
LDN		C061
ANDN		outConter04
STN		resANB_C
									
(*■OR_T命令*)
LD		inTimer06
ST		TON_6.IN
LD		TIME#30s
ST		TON_6.PT
CAL		TON_6
LD		TON_6.Q
ST		outTimer06
LD		TON_6.ET
ST		passed06
									
LD		C065
OR		outTimer06
ST		resOR_T
									
(*■OR_C命令*)
LD		inCounter05
ST		CTU_5.CU
LD		enableCnt
ST		CTU_5.RESET
LD		INT#5000
ST		CTU_5.PV
CAL		CTU_5
LD		CTU_5.Q
ST		outCounter05
LD		CTU_5.CV
ST		valCounter05
									
LD		C069
OR		outCounter05
ST		resOR_C
									
(*■ORB_T命令*)
LD		inTimer07
ST		TON_7.IN
LD		TIME#30s
ST		TON_7.PT
CAL		TON_7
LD		TON_7.Q
ST		outTimer07
LD		TON_7.ET
ST		passed07
									
LD		C075
ORN		outTimer07
STN		resORB_T
									
(*■ORB_C命令*)
LD		inCounter06
ST		CTU_6.CU
LD		enableCnt
ST		CTU_6.RESET
LD		INT#5000
ST		CTU_6.PV
CAL		CTU_6
LD		CTU_6.Q
ST		outCounter06
LD		CTU_6.CV
ST		valCounter06
									
LD		C078
ORN		outCounter06
STN		resORB_C
									
(*■ANL命令*)
LD		input01
OR		C083
ST		IL変数_21
LD		input01
OR		C085
AND		IL変数_21
ST		resANL
									
(*■ORL命令*)
LD		input01
AND		input01
ST		IL変数_22
LD		C089
AND		C091
OR		IL変数_22
ST		resORL
									
(*■MPS、MPP、MRD命令*)
LD		setten0101
AND		setten0102
ST		IL変数_23
LD		IL変数_23
AND		setten0103
ST		IL変数_24
LD		IL変数_24
AND		setten0104
ST		resCoil01
LD		IL変数_24
AND		setten0204
ST		resCoil02
LD		IL変数_24
AND		setten0304
ST		resCoil03
LD		IL変数_23
AND		setten0403
ST		resCoil04
LD		IL変数_23
AND		setten0503
ST		resCoil05
LD		IL変数_23
AND		setten0603
ST		resCoil06
									
LD		setten0101
AND		setten0702
ST		resCoil07
									
LD		setten0101
AND		setten0802
ST		resCoil08
									
LD		setten0101
AND		setten0902
ST		resCoil09
									
(*■ビアメカ問題発生ロジック*)
LD		inBia0102
OR		inBia0202
AND		inBia0101
ST		resBia01
LD		resBia01
AND		inBia0203
ST		resBia02
LD		inBIa0404
OR		inBIa0504
ST		IL変数_25
LD		resBia01
AND		inBia0303
AND		IL変数_25
ST		resBia03
									
(*■CLR命令*)
(*実行されるパターン*)
LD		inCLR01
ST		resCLR01
									
LD		inCLR02
ST		resCLR02
									
(*実行されないパターン*)
LD		inCLR03
ST		resCLR03
AND		inCLR0401
AND		inCLR0402
ST		resCLR04
									
(*■DIFU(TRIGON)命令*)
LD		inDIFU
ST		R_TRIG_1.CLK
CAL		R_TRIG_1
LD		R_TRIG_1.Q
ST		outDIFU
									
LD		outDIFU
OR		holdDIFU
ST		holdDIFU
									
LDN		outDIFU
AND		holdDIFU
ST		resDIFU
									
(*■DIFD(TRIGOFF)命令*)
LD		inDIFD
ST		F_TRIG_1.CLK
CAL		F_TRIG_1
LD		F_TRIG_1.Q
ST		outDIFD
									
LD		outDIFD
OR		holdDIFD
ST		holdDIFD
									
(*-----ここまで-----------------------------------------------------
*)
LD		holdDIFD
ANDN		outDIFD
ST		resDIFD
									
								
							
						
					
						
							
								
							
							
								(*■LD命令*)
LD		input01
ST		resLD
									
(*■LDB命令*)
LDN		input01
STN		resLDB
									
(*■AND命令*)
LDN		C005
AND		input01
ST		resAND
									
(*■ANB命令*)
LDN		C007
ANDN		input01
STN		resANB
									
(*■OR命令*)
LD		C010
OR		input01
ST		resOR
									
(*■ORB命令*)
LD		C015
ORN		input01
STN		resORB
									
(*■OUT命令*)
LD		input01
ST		resOUT
									
(*■OUB命令*)
LDN		input01
STN		resOUB
									
(*■SET命令*)
LD		input01
ANDN		resSET
S		resSET
									
(*■RES命令*)
LD		input01
S		C024
									
LD		input01
R		C024
									
LDN		C024
ST		resRES
									
(*■LD_T命令*)
LD		inTIMER01
ST		TON_1.IN
ST		TON_2.IN
LD		TIME#30s
ST		TON_1.PT
CAL		TON_1
LD		TON_1.Q
ST		resTimer01
LD		TON_1.ET
ST		passed01
LD		TIME#1m
ST		TON_2.PT
CAL		TON_2
LD		TON_2.Q
ST		resTimer02
LD		TON_2.ET
ST		passed02
									
LD		resTimer01
ST		resLD_T01
									
LD		resTimer02
ST		resLD_T02
									
(*■LD_C命令*)
LD		inCounter
ST		CTU_1.CU
LD		enableCnt
ST		CTU_1.RESET
LD		INT#5000
ST		CTU_1.PV
CAL		CTU_1
LD		CTU_1.Q
ST		outConter
LD		CTU_1.CV
ST		valCounter
									
LD		outConter
ST		resLD_C
									
(*■LDB_T命令*)
LD		inTimER02
ST		TON_3.IN
LD		TIME#30s
ST		TON_3.PT
CAL		TON_3
LD		TON_3.Q
ST		resT5
LD		TON_3.ET
ST		passed03
									
LDN		resT5
STN		resLDB_T
									
(*■LDB_C命令*)
LD		inCounter2
ST		CTU_2.CU
LD		enableCnt
ST		CTU_2.RESET
LD		INT#5000
ST		CTU_2.PV
CAL		CTU_2
LD		CTU_2.Q
ST		outConter2
LD		CTU_2.CV
ST		valCounter2
									
LDN		outConter2
STN		resLDB_C
									
(*■AND_T命令*)
LD		inTimeR03
ST		TON_4.IN
LD		TIME#30s
ST		TON_4.PT
CAL		TON_4
LD		TON_4.Q
ST		outTimer
LD		TON_4.ET
ST		passed04
									
LDN		C046
AND		outTimer
ST		resAND_T
									
(*■AND_C命令*)
LD		inCounter3
ST		CTU_3.CU
LD		enableCnt
ST		CTU_3.RESET
LD		INT#5000
ST		CTU_3.PV
CAL		CTU_3
LD		CTU_3.Q
ST		outCounter3
LD		CTU_3.CV
ST		valCounter3
									
LDN		C052
AND		outCounter3
ST		resAND_C
									
(*■ANB_T命令*)
LD		inTimer05
ST		TON_5.IN
LD		TIME#30s
ST		TON_5.PT
CAL		TON_5
LD		TON_5.Q
ST		outTimer05
LD		TON_5.ET
ST		passed05
									
LDN		C055
ANDN		outTimer05
STN		resANB_T
									
(*■ANB_C命令*)
LD		inCounter04
ST		CTU_4.CU
LD		enableCnt
ST		CTU_4.RESET
LD		INT#5000
ST		CTU_4.PV
CAL		CTU_4
LD		CTU_4.Q
ST		outConter04
LD		CTU_4.CV
ST		valCounter04
									
LDN		C061
ANDN		outConter04
STN		resANB_C
									
(*■OR_T命令*)
LD		inTimer06
ST		TON_6.IN
LD		TIME#30s
ST		TON_6.PT
CAL		TON_6
LD		TON_6.Q
ST		outTimer06
LD		TON_6.ET
ST		passed06
									
LD		C065
OR		outTimer06
ST		resOR_T
									
(*■OR_C命令*)
LD		inCounter05
ST		CTU_5.CU
LD		enableCnt
ST		CTU_5.RESET
LD		INT#5000
ST		CTU_5.PV
CAL		CTU_5
LD		CTU_5.Q
ST		outCounter05
LD		CTU_5.CV
ST		valCounter05
									
LD		C069
OR		outCounter05
ST		resOR_C
									
(*■ORB_T命令*)
LD		inTimer07
ST		TON_7.IN
LD		TIME#30s
ST		TON_7.PT
CAL		TON_7
LD		TON_7.Q
ST		outTimer07
LD		TON_7.ET
ST		passed07
									
LD		C075
ORN		outTimer07
STN		resORB_T
									
(*■ORB_C命令*)
LD		inCounter06
ST		CTU_6.CU
LD		enableCnt
ST		CTU_6.RESET
LD		INT#5000
ST		CTU_6.PV
CAL		CTU_6
LD		CTU_6.Q
ST		outCounter06
LD		CTU_6.CV
ST		valCounter06
									
LD		C078
ORN		outCounter06
STN		resORB_C
									
(*■ANL命令*)
LD		input01
OR		C083
ST		IL変数_26
LD		input01
OR		C085
AND		IL変数_26
ST		resANL
									
(*■ORL命令*)
LD		input01
AND		input01
ST		IL変数_27
LD		C089
AND		C091
OR		IL変数_27
ST		resORL
									
(*■MPS、MPP、MRD命令*)
LD		setten0101
AND		setten0102
ST		IL変数_28
LD		IL変数_28
AND		setten0103
ST		IL変数_29
LD		IL変数_29
AND		setten0104
ST		resCoil01
LD		IL変数_29
AND		setten0204
ST		resCoil02
LD		IL変数_29
AND		setten0304
ST		resCoil03
LD		IL変数_28
AND		setten0403
ST		resCoil04
LD		IL変数_28
AND		setten0503
ST		resCoil05
LD		IL変数_28
AND		setten0603
ST		resCoil06
									
LD		setten0101
AND		setten0702
ST		resCoil07
									
LD		setten0101
AND		setten0802
ST		resCoil08
									
LD		setten0101
AND		setten0902
ST		resCoil09
									
(*■ビアメカ問題発生ロジック*)
LD		inBia0102
OR		inBia0202
AND		inBia0101
ST		resBia01
LD		resBia01
AND		inBia0203
ST		resBia02
LD		inBIa0404
OR		inBIa0504
ST		IL変数_30
LD		resBia01
AND		inBia0303
AND		IL変数_30
ST		resBia03
									
(*■CLR命令*)
(*実行されるパターン*)
LD		inCLR01
ST		resCLR01
									
LD		inCLR02
ST		resCLR02
									
(*実行されないパターン*)
LD		inCLR03
ST		resCLR03
AND		inCLR0401
AND		inCLR0402
ST		resCLR04
									
(*■DIFU(TRIGON)命令*)
LD		inDIFU
ST		R_TRIG_1.CLK
CAL		R_TRIG_1
LD		R_TRIG_1.Q
ST		outDIFU
									
LD		outDIFU
OR		holdDIFU
ST		holdDIFU
									
LDN		outDIFU
AND		holdDIFU
ST		resDIFU
									
(*■DIFD(TRIGOFF)命令*)
LD		inDIFD
ST		F_TRIG_1.CLK
CAL		F_TRIG_1
LD		F_TRIG_1.Q
ST		outDIFD
									
LD		outDIFD
OR		holdDIFD
ST		holdDIFD
									
(*-----ここまで-----------------------------------------------------
*)
LD		holdDIFD
ANDN		outDIFD
ST		resDIFD
									
								
							
						
					
						
							
								
							
							
								(*■LD命令*)
LD		input01
ST		resLD
									
(*■LDB命令*)
LDN		input01
STN		resLDB
									
(*■AND命令*)
LDN		C005
AND		input01
ST		resAND
									
(*■ANB命令*)
LDN		C007
ANDN		input01
STN		resANB
									
(*■OR命令*)
LD		C010
OR		input01
ST		resOR
									
(*■ORB命令*)
LD		C015
ORN		input01
STN		resORB
									
(*■OUT命令*)
LD		input01
ST		resOUT
									
(*■OUB命令*)
LDN		input01
STN		resOUB
									
(*■SET命令*)
LD		input01
ANDN		resSET
S		resSET
									
(*■RES命令*)
LD		input01
S		C024
									
LD		input01
R		C024
									
LDN		C024
ST		resRES
									
(*■LD_T命令*)
LD		inTIMER01
ST		TON_1.IN
ST		TON_2.IN
LD		TIME#30s
ST		TON_1.PT
CAL		TON_1
LD		TON_1.Q
ST		resTimer01
LD		TON_1.ET
ST		passed01
LD		TIME#1m
ST		TON_2.PT
CAL		TON_2
LD		TON_2.Q
ST		resTimer02
LD		TON_2.ET
ST		passed02
									
LD		resTimer01
ST		resLD_T01
									
LD		resTimer02
ST		resLD_T02
									
(*■LD_C命令*)
LD		inCounter
ST		CTU_1.CU
LD		enableCnt
ST		CTU_1.RESET
LD		INT#5000
ST		CTU_1.PV
CAL		CTU_1
LD		CTU_1.Q
ST		outConter
LD		CTU_1.CV
ST		valCounter
									
LD		outConter
ST		resLD_C
									
(*■LDB_T命令*)
LD		inTimER02
ST		TON_3.IN
LD		TIME#30s
ST		TON_3.PT
CAL		TON_3
LD		TON_3.Q
ST		resT5
LD		TON_3.ET
ST		passed03
									
LDN		resT5
STN		resLDB_T
									
(*■LDB_C命令*)
LD		inCounter2
ST		CTU_2.CU
LD		enableCnt
ST		CTU_2.RESET
LD		INT#5000
ST		CTU_2.PV
CAL		CTU_2
LD		CTU_2.Q
ST		outConter2
LD		CTU_2.CV
ST		valCounter2
									
LDN		outConter2
STN		resLDB_C
									
(*■AND_T命令*)
LD		inTimeR03
ST		TON_4.IN
LD		TIME#30s
ST		TON_4.PT
CAL		TON_4
LD		TON_4.Q
ST		outTimer
LD		TON_4.ET
ST		passed04
									
LDN		C046
AND		outTimer
ST		resAND_T
									
(*■AND_C命令*)
LD		inCounter3
ST		CTU_3.CU
LD		enableCnt
ST		CTU_3.RESET
LD		INT#5000
ST		CTU_3.PV
CAL		CTU_3
LD		CTU_3.Q
ST		outCounter3
LD		CTU_3.CV
ST		valCounter3
									
LDN		C052
AND		outCounter3
ST		resAND_C
									
(*■ANB_T命令*)
LD		inTimer05
ST		TON_5.IN
LD		TIME#30s
ST		TON_5.PT
CAL		TON_5
LD		TON_5.Q
ST		outTimer05
LD		TON_5.ET
ST		passed05
									
LDN		C055
ANDN		outTimer05
STN		resANB_T
									
(*■ANB_C命令*)
LD		inCounter04
ST		CTU_4.CU
LD		enableCnt
ST		CTU_4.RESET
LD		INT#5000
ST		CTU_4.PV
CAL		CTU_4
LD		CTU_4.Q
ST		outConter04
LD		CTU_4.CV
ST		valCounter04
									
LDN		C061
ANDN		outConter04
STN		resANB_C
									
(*■OR_T命令*)
LD		inTimer06
ST		TON_6.IN
LD		TIME#30s
ST		TON_6.PT
CAL		TON_6
LD		TON_6.Q
ST		outTimer06
LD		TON_6.ET
ST		passed06
									
LD		C065
OR		outTimer06
ST		resOR_T
									
(*■OR_C命令*)
LD		inCounter05
ST		CTU_5.CU
LD		enableCnt
ST		CTU_5.RESET
LD		INT#5000
ST		CTU_5.PV
CAL		CTU_5
LD		CTU_5.Q
ST		outCounter05
LD		CTU_5.CV
ST		valCounter05
									
LD		C069
OR		outCounter05
ST		resOR_C
									
(*■ORB_T命令*)
LD		inTimer07
ST		TON_7.IN
LD		TIME#30s
ST		TON_7.PT
CAL		TON_7
LD		TON_7.Q
ST		outTimer07
LD		TON_7.ET
ST		passed07
									
LD		C075
ORN		outTimer07
STN		resORB_T
									
(*■ORB_C命令*)
LD		inCounter06
ST		CTU_6.CU
LD		enableCnt
ST		CTU_6.RESET
LD		INT#5000
ST		CTU_6.PV
CAL		CTU_6
LD		CTU_6.Q
ST		outCounter06
LD		CTU_6.CV
ST		valCounter06
									
LD		C078
ORN		outCounter06
STN		resORB_C
									
(*■ANL命令*)
LD		input01
OR		C083
ST		IL変数_31
LD		input01
OR		C085
AND		IL変数_31
ST		resANL
									
(*■ORL命令*)
LD		input01
AND		input01
ST		IL変数_32
LD		C089
AND		C091
OR		IL変数_32
ST		resORL
									
(*■MPS、MPP、MRD命令*)
LD		setten0101
AND		setten0102
ST		IL変数_33
LD		IL変数_33
AND		setten0103
ST		IL変数_34
LD		IL変数_34
AND		setten0104
ST		resCoil01
LD		IL変数_34
AND		setten0204
ST		resCoil02
LD		IL変数_34
AND		setten0304
ST		resCoil03
LD		IL変数_33
AND		setten0403
ST		resCoil04
LD		IL変数_33
AND		setten0503
ST		resCoil05
LD		IL変数_33
AND		setten0603
ST		resCoil06
									
LD		setten0101
AND		setten0702
ST		resCoil07
									
LD		setten0101
AND		setten0802
ST		resCoil08
									
LD		setten0101
AND		setten0902
ST		resCoil09
									
(*■ビアメカ問題発生ロジック*)
LD		inBia0102
OR		inBia0202
AND		inBia0101
ST		resBia01
LD		resBia01
AND		inBia0203
ST		resBia02
LD		inBIa0404
OR		inBIa0504
ST		IL変数_35
LD		resBia01
AND		inBia0303
AND		IL変数_35
ST		resBia03
									
(*■CLR命令*)
(*実行されるパターン*)
LD		inCLR01
ST		resCLR01
									
LD		inCLR02
ST		resCLR02
									
(*実行されないパターン*)
LD		inCLR03
ST		resCLR03
AND		inCLR0401
AND		inCLR0402
ST		resCLR04
									
(*■DIFU(TRIGON)命令*)
LD		inDIFU
ST		R_TRIG_1.CLK
CAL		R_TRIG_1
LD		R_TRIG_1.Q
ST		outDIFU
									
LD		outDIFU
OR		holdDIFU
ST		holdDIFU
									
LDN		outDIFU
AND		holdDIFU
ST		resDIFU
									
(*■DIFD(TRIGOFF)命令*)
LD		inDIFD
ST		F_TRIG_1.CLK
CAL		F_TRIG_1
LD		F_TRIG_1.Q
ST		outDIFD
									
LD		outDIFD
OR		holdDIFD
ST		holdDIFD
									
(*-----ここまで-----------------------------------------------------
*)
LD		holdDIFD
ANDN		outDIFD
ST		resDIFD
									
								
							
						
					
						
							
								
							
							
								(*■LD命令*)
LD		input01
ST		resLD
									
(*■LDB命令*)
LDN		input01
STN		resLDB
									
(*■AND命令*)
LDN		C005
AND		input01
ST		resAND
									
(*■ANB命令*)
LDN		C007
ANDN		input01
STN		resANB
									
(*■OR命令*)
LD		C010
OR		input01
ST		resOR
									
(*■ORB命令*)
LD		C015
ORN		input01
STN		resORB
									
(*■OUT命令*)
LD		input01
ST		resOUT
									
(*■OUB命令*)
LDN		input01
STN		resOUB
									
(*■SET命令*)
LD		input01
ANDN		resSET
S		resSET
									
(*■RES命令*)
LD		input01
S		C024
									
LD		input01
R		C024
									
LDN		C024
ST		resRES
									
(*■LD_T命令*)
LD		inTIMER01
ST		TON_1.IN
ST		TON_2.IN
LD		TIME#30s
ST		TON_1.PT
CAL		TON_1
LD		TON_1.Q
ST		resTimer01
LD		TON_1.ET
ST		passed01
LD		TIME#1m
ST		TON_2.PT
CAL		TON_2
LD		TON_2.Q
ST		resTimer02
LD		TON_2.ET
ST		passed02
									
LD		resTimer01
ST		resLD_T01
									
LD		resTimer02
ST		resLD_T02
									
(*■LD_C命令*)
LD		inCounter
ST		CTU_1.CU
LD		enableCnt
ST		CTU_1.RESET
LD		INT#5000
ST		CTU_1.PV
CAL		CTU_1
LD		CTU_1.Q
ST		outConter
LD		CTU_1.CV
ST		valCounter
									
LD		outConter
ST		resLD_C
									
(*■LDB_T命令*)
LD		inTimER02
ST		TON_3.IN
LD		TIME#30s
ST		TON_3.PT
CAL		TON_3
LD		TON_3.Q
ST		resT5
LD		TON_3.ET
ST		passed03
									
LDN		resT5
STN		resLDB_T
									
(*■LDB_C命令*)
LD		inCounter2
ST		CTU_2.CU
LD		enableCnt
ST		CTU_2.RESET
LD		INT#5000
ST		CTU_2.PV
CAL		CTU_2
LD		CTU_2.Q
ST		outConter2
LD		CTU_2.CV
ST		valCounter2
									
LDN		outConter2
STN		resLDB_C
									
(*■AND_T命令*)
LD		inTimeR03
ST		TON_4.IN
LD		TIME#30s
ST		TON_4.PT
CAL		TON_4
LD		TON_4.Q
ST		outTimer
LD		TON_4.ET
ST		passed04
									
LDN		C046
AND		outTimer
ST		resAND_T
									
(*■AND_C命令*)
LD		inCounter3
ST		CTU_3.CU
LD		enableCnt
ST		CTU_3.RESET
LD		INT#5000
ST		CTU_3.PV
CAL		CTU_3
LD		CTU_3.Q
ST		outCounter3
LD		CTU_3.CV
ST		valCounter3
									
LDN		C052
AND		outCounter3
ST		resAND_C
									
(*■ANB_T命令*)
LD		inTimer05
ST		TON_5.IN
LD		TIME#30s
ST		TON_5.PT
CAL		TON_5
LD		TON_5.Q
ST		outTimer05
LD		TON_5.ET
ST		passed05
									
LDN		C055
ANDN		outTimer05
STN		resANB_T
									
(*■ANB_C命令*)
LD		inCounter04
ST		CTU_4.CU
LD		enableCnt
ST		CTU_4.RESET
LD		INT#5000
ST		CTU_4.PV
CAL		CTU_4
LD		CTU_4.Q
ST		outConter04
LD		CTU_4.CV
ST		valCounter04
									
LDN		C061
ANDN		outConter04
STN		resANB_C
									
(*■OR_T命令*)
LD		inTimer06
ST		TON_6.IN
LD		TIME#30s
ST		TON_6.PT
CAL		TON_6
LD		TON_6.Q
ST		outTimer06
LD		TON_6.ET
ST		passed06
									
LD		C065
OR		outTimer06
ST		resOR_T
									
(*■OR_C命令*)
LD		inCounter05
ST		CTU_5.CU
LD		enableCnt
ST		CTU_5.RESET
LD		INT#5000
ST		CTU_5.PV
CAL		CTU_5
LD		CTU_5.Q
ST		outCounter05
LD		CTU_5.CV
ST		valCounter05
									
LD		C069
OR		outCounter05
ST		resOR_C
									
(*■ORB_T命令*)
LD		inTimer07
ST		TON_7.IN
LD		TIME#30s
ST		TON_7.PT
CAL		TON_7
LD		TON_7.Q
ST		outTimer07
LD		TON_7.ET
ST		passed07
									
LD		C075
ORN		outTimer07
STN		resORB_T
									
(*■ORB_C命令*)
LD		inCounter06
ST		CTU_6.CU
LD		enableCnt
ST		CTU_6.RESET
LD		INT#5000
ST		CTU_6.PV
CAL		CTU_6
LD		CTU_6.Q
ST		outCounter06
LD		CTU_6.CV
ST		valCounter06
									
LD		C078
ORN		outCounter06
STN		resORB_C
									
(*■ANL命令*)
LD		input01
OR		C083
ST		IL変数_36
LD		input01
OR		C085
AND		IL変数_36
ST		resANL
									
(*■ORL命令*)
LD		input01
AND		input01
ST		IL変数_37
LD		C089
AND		C091
OR		IL変数_37
ST		resORL
									
(*■MPS、MPP、MRD命令*)
LD		setten0101
AND		setten0102
ST		IL変数_38
LD		IL変数_38
AND		setten0103
ST		IL変数_39
LD		IL変数_39
AND		setten0104
ST		resCoil01
LD		IL変数_39
AND		setten0204
ST		resCoil02
LD		IL変数_39
AND		setten0304
ST		resCoil03
LD		IL変数_38
AND		setten0403
ST		resCoil04
LD		IL変数_38
AND		setten0503
ST		resCoil05
LD		IL変数_38
AND		setten0603
ST		resCoil06
									
LD		setten0101
AND		setten0702
ST		resCoil07
									
LD		setten0101
AND		setten0802
ST		resCoil08
									
LD		setten0101
AND		setten0902
ST		resCoil09
									
(*■ビアメカ問題発生ロジック*)
LD		inBia0102
OR		inBia0202
AND		inBia0101
ST		resBia01
LD		resBia01
AND		inBia0203
ST		resBia02
LD		inBIa0404
OR		inBIa0504
ST		IL変数_40
LD		resBia01
AND		inBia0303
AND		IL変数_40
ST		resBia03
									
(*■CLR命令*)
(*実行されるパターン*)
LD		inCLR01
ST		resCLR01
									
LD		inCLR02
ST		resCLR02
									
(*実行されないパターン*)
LD		inCLR03
ST		resCLR03
AND		inCLR0401
AND		inCLR0402
ST		resCLR04
									
(*■DIFU(TRIGON)命令*)
LD		inDIFU
ST		R_TRIG_1.CLK
CAL		R_TRIG_1
LD		R_TRIG_1.Q
ST		outDIFU
									
LD		outDIFU
OR		holdDIFU
ST		holdDIFU
									
LDN		outDIFU
AND		holdDIFU
ST		resDIFU
									
(*■DIFD(TRIGOFF)命令*)
LD		inDIFD
ST		F_TRIG_1.CLK
CAL		F_TRIG_1
LD		F_TRIG_1.Q
ST		outDIFD
									
LD		outDIFD
OR		holdDIFD
ST		holdDIFD
									
(*-----ここまで-----------------------------------------------------
*)
LD		holdDIFD
ANDN		outDIFD
ST		resDIFD
									
								
							
						
					
						
							
								
							
							
								(*■LD命令*)
LD		input01
ST		resLD
									
(*■LDB命令*)
LDN		input01
STN		resLDB
									
(*■AND命令*)
LDN		C005
AND		input01
ST		resAND
									
(*■ANB命令*)
LDN		C007
ANDN		input01
STN		resANB
									
(*■OR命令*)
LD		C010
OR		input01
ST		resOR
									
(*■ORB命令*)
LD		C015
ORN		input01
STN		resORB
									
(*■OUT命令*)
LD		input01
ST		resOUT
									
(*■OUB命令*)
LDN		input01
STN		resOUB
									
(*■SET命令*)
LD		input01
ANDN		resSET
S		resSET
									
(*■RES命令*)
LD		input01
S		C024
									
LD		input01
R		C024
									
LDN		C024
ST		resRES
									
(*■LD_T命令*)
LD		inTIMER01
ST		TON_1.IN
ST		TON_2.IN
LD		TIME#30s
ST		TON_1.PT
CAL		TON_1
LD		TON_1.Q
ST		resTimer01
LD		TON_1.ET
ST		passed01
LD		TIME#1m
ST		TON_2.PT
CAL		TON_2
LD		TON_2.Q
ST		resTimer02
LD		TON_2.ET
ST		passed02
									
LD		resTimer01
ST		resLD_T01
									
LD		resTimer02
ST		resLD_T02
									
(*■LD_C命令*)
LD		inCounter
ST		CTU_1.CU
LD		enableCnt
ST		CTU_1.RESET
LD		INT#5000
ST		CTU_1.PV
CAL		CTU_1
LD		CTU_1.Q
ST		outConter
LD		CTU_1.CV
ST		valCounter
									
LD		outConter
ST		resLD_C
									
(*■LDB_T命令*)
LD		inTimER02
ST		TON_3.IN
LD		TIME#30s
ST		TON_3.PT
CAL		TON_3
LD		TON_3.Q
ST		resT5
LD		TON_3.ET
ST		passed03
									
LDN		resT5
STN		resLDB_T
									
(*■LDB_C命令*)
LD		inCounter2
ST		CTU_2.CU
LD		enableCnt
ST		CTU_2.RESET
LD		INT#5000
ST		CTU_2.PV
CAL		CTU_2
LD		CTU_2.Q
ST		outConter2
LD		CTU_2.CV
ST		valCounter2
									
LDN		outConter2
STN		resLDB_C
									
(*■AND_T命令*)
LD		inTimeR03
ST		TON_4.IN
LD		TIME#30s
ST		TON_4.PT
CAL		TON_4
LD		TON_4.Q
ST		outTimer
LD		TON_4.ET
ST		passed04
									
LDN		C046
AND		outTimer
ST		resAND_T
									
(*■AND_C命令*)
LD		inCounter3
ST		CTU_3.CU
LD		enableCnt
ST		CTU_3.RESET
LD		INT#5000
ST		CTU_3.PV
CAL		CTU_3
LD		CTU_3.Q
ST		outCounter3
LD		CTU_3.CV
ST		valCounter3
									
LDN		C052
AND		outCounter3
ST		resAND_C
									
(*■ANB_T命令*)
LD		inTimer05
ST		TON_5.IN
LD		TIME#30s
ST		TON_5.PT
CAL		TON_5
LD		TON_5.Q
ST		outTimer05
LD		TON_5.ET
ST		passed05
									
LDN		C055
ANDN		outTimer05
STN		resANB_T
									
(*■ANB_C命令*)
LD		inCounter04
ST		CTU_4.CU
LD		enableCnt
ST		CTU_4.RESET
LD		INT#5000
ST		CTU_4.PV
CAL		CTU_4
LD		CTU_4.Q
ST		outConter04
LD		CTU_4.CV
ST		valCounter04
									
LDN		C061
ANDN		outConter04
STN		resANB_C
									
(*■OR_T命令*)
LD		inTimer06
ST		TON_6.IN
LD		TIME#30s
ST		TON_6.PT
CAL		TON_6
LD		TON_6.Q
ST		outTimer06
LD		TON_6.ET
ST		passed06
									
LD		C065
OR		outTimer06
ST		resOR_T
									
(*■OR_C命令*)
LD		inCounter05
ST		CTU_5.CU
LD		enableCnt
ST		CTU_5.RESET
LD		INT#5000
ST		CTU_5.PV
CAL		CTU_5
LD		CTU_5.Q
ST		outCounter05
LD		CTU_5.CV
ST		valCounter05
									
LD		C069
OR		outCounter05
ST		resOR_C
									
(*■ORB_T命令*)
LD		inTimer07
ST		TON_7.IN
LD		TIME#30s
ST		TON_7.PT
CAL		TON_7
LD		TON_7.Q
ST		outTimer07
LD		TON_7.ET
ST		passed07
									
LD		C075
ORN		outTimer07
STN		resORB_T
									
(*■ORB_C命令*)
LD		inCounter06
ST		CTU_6.CU
LD		enableCnt
ST		CTU_6.RESET
LD		INT#5000
ST		CTU_6.PV
CAL		CTU_6
LD		CTU_6.Q
ST		outCounter06
LD		CTU_6.CV
ST		valCounter06
									
LD		C078
ORN		outCounter06
STN		resORB_C
									
(*■ANL命令*)
LD		input01
OR		C083
ST		IL変数_41
LD		input01
OR		C085
AND		IL変数_41
ST		resANL
									
(*■ORL命令*)
LD		input01
AND		input01
ST		IL変数_42
LD		C089
AND		C091
OR		IL変数_42
ST		resORL
									
(*■MPS、MPP、MRD命令*)
LD		setten0101
AND		setten0102
ST		IL変数_43
LD		IL変数_43
AND		setten0103
ST		IL変数_44
LD		IL変数_44
AND		setten0104
ST		resCoil01
LD		IL変数_44
AND		setten0204
ST		resCoil02
LD		IL変数_44
AND		setten0304
ST		resCoil03
LD		IL変数_43
AND		setten0403
ST		resCoil04
LD		IL変数_43
AND		setten0503
ST		resCoil05
LD		IL変数_43
AND		setten0603
ST		resCoil06
									
LD		setten0101
AND		setten0702
ST		resCoil07
									
LD		setten0101
AND		setten0802
ST		resCoil08
									
LD		setten0101
AND		setten0902
ST		resCoil09
									
(*■ビアメカ問題発生ロジック*)
LD		inBia0102
OR		inBia0202
AND		inBia0101
ST		resBia01
LD		resBia01
AND		inBia0203
ST		resBia02
LD		inBIa0404
OR		inBIa0504
ST		IL変数_45
LD		resBia01
AND		inBia0303
AND		IL変数_45
ST		resBia03
									
(*■CLR命令*)
(*実行されるパターン*)
LD		inCLR01
ST		resCLR01
									
LD		inCLR02
ST		resCLR02
									
(*実行されないパターン*)
LD		inCLR03
ST		resCLR03
AND		inCLR0401
AND		inCLR0402
ST		resCLR04
									
(*■DIFU(TRIGON)命令*)
LD		inDIFU
ST		R_TRIG_1.CLK
CAL		R_TRIG_1
LD		R_TRIG_1.Q
ST		outDIFU
									
LD		outDIFU
OR		holdDIFU
ST		holdDIFU
									
LDN		outDIFU
AND		holdDIFU
ST		resDIFU
									
(*■DIFD(TRIGOFF)命令*)
LD		inDIFD
ST		F_TRIG_1.CLK
CAL		F_TRIG_1
LD		F_TRIG_1.Q
ST		outDIFD
									
LD		outDIFD
OR		holdDIFD
ST		holdDIFD
									
(*-----ここまで-----------------------------------------------------
*)
LD		holdDIFD
ANDN		outDIFD
ST		resDIFD
									
								
							
						
					
						
							
								
							
							
								(*■LD命令*)
LD		input01
ST		resLD
									
(*■LDB命令*)
LDN		input01
STN		resLDB
									
(*■AND命令*)
LDN		C005
AND		input01
ST		resAND
									
(*■ANB命令*)
LDN		C007
ANDN		input01
STN		resANB
									
(*■OR命令*)
LD		C010
OR		input01
ST		resOR
									
(*■ORB命令*)
LD		C015
ORN		input01
STN		resORB
									
(*■OUT命令*)
LD		input01
ST		resOUT
									
(*■OUB命令*)
LDN		input01
STN		resOUB
									
(*■SET命令*)
LD		input01
ANDN		resSET
S		resSET
									
(*■RES命令*)
LD		input01
S		C024
									
LD		input01
R		C024
									
LDN		C024
ST		resRES
									
(*■LD_T命令*)
LD		inTIMER01
ST		TON_1.IN
ST		TON_2.IN
LD		TIME#30s
ST		TON_1.PT
CAL		TON_1
LD		TON_1.Q
ST		resTimer01
LD		TON_1.ET
ST		passed01
LD		TIME#1m
ST		TON_2.PT
CAL		TON_2
LD		TON_2.Q
ST		resTimer02
LD		TON_2.ET
ST		passed02
									
LD		resTimer01
ST		resLD_T01
									
LD		resTimer02
ST		resLD_T02
									
(*■LD_C命令*)
LD		inCounter
ST		CTU_1.CU
LD		enableCnt
ST		CTU_1.RESET
LD		INT#5000
ST		CTU_1.PV
CAL		CTU_1
LD		CTU_1.Q
ST		outConter
LD		CTU_1.CV
ST		valCounter
									
LD		outConter
ST		resLD_C
									
(*■LDB_T命令*)
LD		inTimER02
ST		TON_3.IN
LD		TIME#30s
ST		TON_3.PT
CAL		TON_3
LD		TON_3.Q
ST		resT5
LD		TON_3.ET
ST		passed03
									
LDN		resT5
STN		resLDB_T
									
(*■LDB_C命令*)
LD		inCounter2
ST		CTU_2.CU
LD		enableCnt
ST		CTU_2.RESET
LD		INT#5000
ST		CTU_2.PV
CAL		CTU_2
LD		CTU_2.Q
ST		outConter2
LD		CTU_2.CV
ST		valCounter2
									
LDN		outConter2
STN		resLDB_C
									
(*■AND_T命令*)
LD		inTimeR03
ST		TON_4.IN
LD		TIME#30s
ST		TON_4.PT
CAL		TON_4
LD		TON_4.Q
ST		outTimer
LD		TON_4.ET
ST		passed04
									
LDN		C046
AND		outTimer
ST		resAND_T
									
(*■AND_C命令*)
LD		inCounter3
ST		CTU_3.CU
LD		enableCnt
ST		CTU_3.RESET
LD		INT#5000
ST		CTU_3.PV
CAL		CTU_3
LD		CTU_3.Q
ST		outCounter3
LD		CTU_3.CV
ST		valCounter3
									
LDN		C052
AND		outCounter3
ST		resAND_C
									
(*■ANB_T命令*)
LD		inTimer05
ST		TON_5.IN
LD		TIME#30s
ST		TON_5.PT
CAL		TON_5
LD		TON_5.Q
ST		outTimer05
LD		TON_5.ET
ST		passed05
									
LDN		C055
ANDN		outTimer05
STN		resANB_T
									
(*■ANB_C命令*)
LD		inCounter04
ST		CTU_4.CU
LD		enableCnt
ST		CTU_4.RESET
LD		INT#5000
ST		CTU_4.PV
CAL		CTU_4
LD		CTU_4.Q
ST		outConter04
LD		CTU_4.CV
ST		valCounter04
									
LDN		C061
ANDN		outConter04
STN		resANB_C
									
(*■OR_T命令*)
LD		inTimer06
ST		TON_6.IN
LD		TIME#30s
ST		TON_6.PT
CAL		TON_6
LD		TON_6.Q
ST		outTimer06
LD		TON_6.ET
ST		passed06
									
LD		C065
OR		outTimer06
ST		resOR_T
									
(*■OR_C命令*)
LD		inCounter05
ST		CTU_5.CU
LD		enableCnt
ST		CTU_5.RESET
LD		INT#5000
ST		CTU_5.PV
CAL		CTU_5
LD		CTU_5.Q
ST		outCounter05
LD		CTU_5.CV
ST		valCounter05
									
LD		C069
OR		outCounter05
ST		resOR_C
									
(*■ORB_T命令*)
LD		inTimer07
ST		TON_7.IN
LD		TIME#30s
ST		TON_7.PT
CAL		TON_7
LD		TON_7.Q
ST		outTimer07
LD		TON_7.ET
ST		passed07
									
LD		C075
ORN		outTimer07
STN		resORB_T
									
(*■ORB_C命令*)
LD		inCounter06
ST		CTU_6.CU
LD		enableCnt
ST		CTU_6.RESET
LD		INT#5000
ST		CTU_6.PV
CAL		CTU_6
LD		CTU_6.Q
ST		outCounter06
LD		CTU_6.CV
ST		valCounter06
									
LD		C078
ORN		outCounter06
STN		resORB_C
									
(*■ANL命令*)
LD		input01
OR		C083
ST		IL変数_46
LD		input01
OR		C085
AND		IL変数_46
ST		resANL
									
(*■ORL命令*)
LD		input01
AND		input01
ST		IL変数_47
LD		C089
AND		C091
OR		IL変数_47
ST		resORL
									
(*■MPS、MPP、MRD命令*)
LD		setten0101
AND		setten0102
ST		IL変数_48
LD		IL変数_48
AND		setten0103
ST		IL変数_49
LD		IL変数_49
AND		setten0104
ST		resCoil01
LD		IL変数_49
AND		setten0204
ST		resCoil02
LD		IL変数_49
AND		setten0304
ST		resCoil03
LD		IL変数_48
AND		setten0403
ST		resCoil04
LD		IL変数_48
AND		setten0503
ST		resCoil05
LD		IL変数_48
AND		setten0603
ST		resCoil06
									
LD		setten0101
AND		setten0702
ST		resCoil07
									
LD		setten0101
AND		setten0802
ST		resCoil08
									
LD		setten0101
AND		setten0902
ST		resCoil09
									
(*■ビアメカ問題発生ロジック*)
LD		inBia0102
OR		inBia0202
AND		inBia0101
ST		resBia01
LD		resBia01
AND		inBia0203
ST		resBia02
LD		inBIa0404
OR		inBIa0504
ST		IL変数_50
LD		resBia01
AND		inBia0303
AND		IL変数_50
ST		resBia03
									
(*■CLR命令*)
(*実行されるパターン*)
LD		inCLR01
ST		resCLR01
									
LD		inCLR02
ST		resCLR02
									
(*実行されないパターン*)
LD		inCLR03
ST		resCLR03
AND		inCLR0401
AND		inCLR0402
ST		resCLR04
									
(*■DIFU(TRIGON)命令*)
LD		inDIFU
ST		R_TRIG_1.CLK
CAL		R_TRIG_1
LD		R_TRIG_1.Q
ST		outDIFU
									
LD		outDIFU
OR		holdDIFU
ST		holdDIFU
									
LDN		outDIFU
AND		holdDIFU
ST		resDIFU
									
(*■DIFD(TRIGOFF)命令*)
LD		inDIFD
ST		F_TRIG_1.CLK
CAL		F_TRIG_1
LD		F_TRIG_1.Q
ST		outDIFD
									
LD		outDIFD
OR		holdDIFD
ST		holdDIFD
									
(*-----ここまで-----------------------------------------------------
*)
LD		holdDIFD
ANDN		outDIFD
ST		resDIFD
									
								
							
						
					
						
							
								
							
							
								(*■LD命令*)
LD		input01
ST		resLD
									
(*■LDB命令*)
LDN		input01
STN		resLDB
									
(*■AND命令*)
LDN		C005
AND		input01
ST		resAND
									
(*■ANB命令*)
LDN		C007
ANDN		input01
STN		resANB
									
(*■OR命令*)
LD		C010
OR		input01
ST		resOR
									
(*■ORB命令*)
LD		C015
ORN		input01
STN		resORB
									
(*■OUT命令*)
LD		input01
ST		resOUT
									
(*■OUB命令*)
LDN		input01
STN		resOUB
									
(*■SET命令*)
LD		input01
ANDN		resSET
S		resSET
									
(*■RES命令*)
LD		input01
S		C024
									
LD		input01
R		C024
									
LDN		C024
ST		resRES
									
(*■LD_T命令*)
LD		inTIMER01
ST		TON_1.IN
ST		TON_2.IN
LD		TIME#30s
ST		TON_1.PT
CAL		TON_1
LD		TON_1.Q
ST		resTimer01
LD		TON_1.ET
ST		passed01
LD		TIME#1m
ST		TON_2.PT
CAL		TON_2
LD		TON_2.Q
ST		resTimer02
LD		TON_2.ET
ST		passed02
									
LD		resTimer01
ST		resLD_T01
									
LD		resTimer02
ST		resLD_T02
									
(*■LD_C命令*)
LD		inCounter
ST		CTU_1.CU
LD		enableCnt
ST		CTU_1.RESET
LD		INT#5000
ST		CTU_1.PV
CAL		CTU_1
LD		CTU_1.Q
ST		outConter
LD		CTU_1.CV
ST		valCounter
									
LD		outConter
ST		resLD_C
									
(*■LDB_T命令*)
LD		inTimER02
ST		TON_3.IN
LD		TIME#30s
ST		TON_3.PT
CAL		TON_3
LD		TON_3.Q
ST		resT5
LD		TON_3.ET
ST		passed03
									
LDN		resT5
STN		resLDB_T
									
(*■LDB_C命令*)
LD		inCounter2
ST		CTU_2.CU
LD		enableCnt
ST		CTU_2.RESET
LD		INT#5000
ST		CTU_2.PV
CAL		CTU_2
LD		CTU_2.Q
ST		outConter2
LD		CTU_2.CV
ST		valCounter2
									
LDN		outConter2
STN		resLDB_C
									
(*■AND_T命令*)
LD		inTimeR03
ST		TON_4.IN
LD		TIME#30s
ST		TON_4.PT
CAL		TON_4
LD		TON_4.Q
ST		outTimer
LD		TON_4.ET
ST		passed04
									
LDN		C046
AND		outTimer
ST		resAND_T
									
(*■AND_C命令*)
LD		inCounter3
ST		CTU_3.CU
LD		enableCnt
ST		CTU_3.RESET
LD		INT#5000
ST		CTU_3.PV
CAL		CTU_3
LD		CTU_3.Q
ST		outCounter3
LD		CTU_3.CV
ST		valCounter3
									
LDN		C052
AND		outCounter3
ST		resAND_C
									
(*■ANB_T命令*)
LD		inTimer05
ST		TON_5.IN
LD		TIME#30s
ST		TON_5.PT
CAL		TON_5
LD		TON_5.Q
ST		outTimer05
LD		TON_5.ET
ST		passed05
									
LDN		C055
ANDN		outTimer05
STN		resANB_T
									
(*■ANB_C命令*)
LD		inCounter04
ST		CTU_4.CU
LD		enableCnt
ST		CTU_4.RESET
LD		INT#5000
ST		CTU_4.PV
CAL		CTU_4
LD		CTU_4.Q
ST		outConter04
LD		CTU_4.CV
ST		valCounter04
									
LDN		C061
ANDN		outConter04
STN		resANB_C
									
(*■OR_T命令*)
LD		inTimer06
ST		TON_6.IN
LD		TIME#30s
ST		TON_6.PT
CAL		TON_6
LD		TON_6.Q
ST		outTimer06
LD		TON_6.ET
ST		passed06
									
LD		C065
OR		outTimer06
ST		resOR_T
									
(*■OR_C命令*)
LD		inCounter05
ST		CTU_5.CU
LD		enableCnt
ST		CTU_5.RESET
LD		INT#5000
ST		CTU_5.PV
CAL		CTU_5
LD		CTU_5.Q
ST		outCounter05
LD		CTU_5.CV
ST		valCounter05
									
LD		C069
OR		outCounter05
ST		resOR_C
									
(*■ORB_T命令*)
LD		inTimer07
ST		TON_7.IN
LD		TIME#30s
ST		TON_7.PT
CAL		TON_7
LD		TON_7.Q
ST		outTimer07
LD		TON_7.ET
ST		passed07
									
LD		C075
ORN		outTimer07
STN		resORB_T
									
(*■ORB_C命令*)
LD		inCounter06
ST		CTU_6.CU
LD		enableCnt
ST		CTU_6.RESET
LD		INT#5000
ST		CTU_6.PV
CAL		CTU_6
LD		CTU_6.Q
ST		outCounter06
LD		CTU_6.CV
ST		valCounter06
									
LD		C078
ORN		outCounter06
STN		resORB_C
									
(*■ANL命令*)
LD		input01
OR		C083
ST		IL変数_51
LD		input01
OR		C085
AND		IL変数_51
ST		resANL
									
(*■ORL命令*)
LD		input01
AND		input01
ST		IL変数_52
LD		C089
AND		C091
OR		IL変数_52
ST		resORL
									
(*■MPS、MPP、MRD命令*)
LD		setten0101
AND		setten0102
ST		IL変数_53
LD		IL変数_53
AND		setten0103
ST		IL変数_54
LD		IL変数_54
AND		setten0104
ST		resCoil01
LD		IL変数_54
AND		setten0204
ST		resCoil02
LD		IL変数_54
AND		setten0304
ST		resCoil03
LD		IL変数_53
AND		setten0403
ST		resCoil04
LD		IL変数_53
AND		setten0503
ST		resCoil05
LD		IL変数_53
AND		setten0603
ST		resCoil06
									
LD		setten0101
AND		setten0702
ST		resCoil07
									
LD		setten0101
AND		setten0802
ST		resCoil08
									
LD		setten0101
AND		setten0902
ST		resCoil09
									
(*■ビアメカ問題発生ロジック*)
LD		inBia0102
OR		inBia0202
AND		inBia0101
ST		resBia01
LD		resBia01
AND		inBia0203
ST		resBia02
LD		inBIa0404
OR		inBIa0504
ST		IL変数_55
LD		resBia01
AND		inBia0303
AND		IL変数_55
ST		resBia03
									
(*■CLR命令*)
(*実行されるパターン*)
LD		inCLR01
ST		resCLR01
									
LD		inCLR02
ST		resCLR02
									
(*実行されないパターン*)
LD		inCLR03
ST		resCLR03
AND		inCLR0401
AND		inCLR0402
ST		resCLR04
									
(*■DIFU(TRIGON)命令*)
LD		inDIFU
ST		R_TRIG_1.CLK
CAL		R_TRIG_1
LD		R_TRIG_1.Q
ST		outDIFU
									
LD		outDIFU
OR		holdDIFU
ST		holdDIFU
									
LDN		outDIFU
AND		holdDIFU
ST		resDIFU
									
(*■DIFD(TRIGOFF)命令*)
LD		inDIFD
ST		F_TRIG_1.CLK
CAL		F_TRIG_1
LD		F_TRIG_1.Q
ST		outDIFD
									
LD		outDIFD
OR		holdDIFD
ST		holdDIFD
									
(*-----ここまで-----------------------------------------------------
*)
LD		holdDIFD
ANDN		outDIFD
ST		resDIFD
									
								
							
						
					
						
							
								
							
							
								(*■LD命令*)
LD		input01
ST		resLD
									
(*■LDB命令*)
LDN		input01
STN		resLDB
									
(*■AND命令*)
LDN		C005
AND		input01
ST		resAND
									
(*■ANB命令*)
LDN		C007
ANDN		input01
STN		resANB
									
(*■OR命令*)
LD		C010
OR		input01
ST		resOR
									
(*■ORB命令*)
LD		C015
ORN		input01
STN		resORB
									
(*■OUT命令*)
LD		input01
ST		resOUT
									
(*■OUB命令*)
LDN		input01
STN		resOUB
									
(*■SET命令*)
LD		input01
ANDN		resSET
S		resSET
									
(*■RES命令*)
LD		input01
S		C024
									
LD		input01
R		C024
									
LDN		C024
ST		resRES
									
(*■LD_T命令*)
LD		inTIMER01
ST		TON_1.IN
ST		TON_2.IN
LD		TIME#30s
ST		TON_1.PT
CAL		TON_1
LD		TON_1.Q
ST		resTimer01
LD		TON_1.ET
ST		passed01
LD		TIME#1m
ST		TON_2.PT
CAL		TON_2
LD		TON_2.Q
ST		resTimer02
LD		TON_2.ET
ST		passed02
									
LD		resTimer01
ST		resLD_T01
									
LD		resTimer02
ST		resLD_T02
									
(*■LD_C命令*)
LD		inCounter
ST		CTU_1.CU
LD		enableCnt
ST		CTU_1.RESET
LD		INT#5000
ST		CTU_1.PV
CAL		CTU_1
LD		CTU_1.Q
ST		outConter
LD		CTU_1.CV
ST		valCounter
									
LD		outConter
ST		resLD_C
									
(*■LDB_T命令*)
LD		inTimER02
ST		TON_3.IN
LD		TIME#30s
ST		TON_3.PT
CAL		TON_3
LD		TON_3.Q
ST		resT5
LD		TON_3.ET
ST		passed03
									
LDN		resT5
STN		resLDB_T
									
(*■LDB_C命令*)
LD		inCounter2
ST		CTU_2.CU
LD		enableCnt
ST		CTU_2.RESET
LD		INT#5000
ST		CTU_2.PV
CAL		CTU_2
LD		CTU_2.Q
ST		outConter2
LD		CTU_2.CV
ST		valCounter2
									
LDN		outConter2
STN		resLDB_C
									
(*■AND_T命令*)
LD		inTimeR03
ST		TON_4.IN
LD		TIME#30s
ST		TON_4.PT
CAL		TON_4
LD		TON_4.Q
ST		outTimer
LD		TON_4.ET
ST		passed04
									
LDN		C046
AND		outTimer
ST		resAND_T
									
(*■AND_C命令*)
LD		inCounter3
ST		CTU_3.CU
LD		enableCnt
ST		CTU_3.RESET
LD		INT#5000
ST		CTU_3.PV
CAL		CTU_3
LD		CTU_3.Q
ST		outCounter3
LD		CTU_3.CV
ST		valCounter3
									
LDN		C052
AND		outCounter3
ST		resAND_C
									
(*■ANB_T命令*)
LD		inTimer05
ST		TON_5.IN
LD		TIME#30s
ST		TON_5.PT
CAL		TON_5
LD		TON_5.Q
ST		outTimer05
LD		TON_5.ET
ST		passed05
									
LDN		C055
ANDN		outTimer05
STN		resANB_T
									
(*■ANB_C命令*)
LD		inCounter04
ST		CTU_4.CU
LD		enableCnt
ST		CTU_4.RESET
LD		INT#5000
ST		CTU_4.PV
CAL		CTU_4
LD		CTU_4.Q
ST		outConter04
LD		CTU_4.CV
ST		valCounter04
									
LDN		C061
ANDN		outConter04
STN		resANB_C
									
(*■OR_T命令*)
LD		inTimer06
ST		TON_6.IN
LD		TIME#30s
ST		TON_6.PT
CAL		TON_6
LD		TON_6.Q
ST		outTimer06
LD		TON_6.ET
ST		passed06
									
LD		C065
OR		outTimer06
ST		resOR_T
									
(*■OR_C命令*)
LD		inCounter05
ST		CTU_5.CU
LD		enableCnt
ST		CTU_5.RESET
LD		INT#5000
ST		CTU_5.PV
CAL		CTU_5
LD		CTU_5.Q
ST		outCounter05
LD		CTU_5.CV
ST		valCounter05
									
LD		C069
OR		outCounter05
ST		resOR_C
									
(*■ORB_T命令*)
LD		inTimer07
ST		TON_7.IN
LD		TIME#30s
ST		TON_7.PT
CAL		TON_7
LD		TON_7.Q
ST		outTimer07
LD		TON_7.ET
ST		passed07
									
LD		C075
ORN		outTimer07
STN		resORB_T
									
(*■ORB_C命令*)
LD		inCounter06
ST		CTU_6.CU
LD		enableCnt
ST		CTU_6.RESET
LD		INT#5000
ST		CTU_6.PV
CAL		CTU_6
LD		CTU_6.Q
ST		outCounter06
LD		CTU_6.CV
ST		valCounter06
									
LD		C078
ORN		outCounter06
STN		resORB_C
									
(*■ANL命令*)
LD		input01
OR		C083
ST		IL変数_56
LD		input01
OR		C085
AND		IL変数_56
ST		resANL
									
(*■ORL命令*)
LD		input01
AND		input01
ST		IL変数_57
LD		C089
AND		C091
OR		IL変数_57
ST		resORL
									
(*■MPS、MPP、MRD命令*)
LD		setten0101
AND		setten0102
ST		IL変数_58
LD		IL変数_58
AND		setten0103
ST		IL変数_59
LD		IL変数_59
AND		setten0104
ST		resCoil01
LD		IL変数_59
AND		setten0204
ST		resCoil02
LD		IL変数_59
AND		setten0304
ST		resCoil03
LD		IL変数_58
AND		setten0403
ST		resCoil04
LD		IL変数_58
AND		setten0503
ST		resCoil05
LD		IL変数_58
AND		setten0603
ST		resCoil06
									
LD		setten0101
AND		setten0702
ST		resCoil07
									
LD		setten0101
AND		setten0802
ST		resCoil08
									
LD		setten0101
AND		setten0902
ST		resCoil09
									
(*■ビアメカ問題発生ロジック*)
LD		inBia0102
OR		inBia0202
AND		inBia0101
ST		resBia01
LD		resBia01
AND		inBia0203
ST		resBia02
LD		inBIa0404
OR		inBIa0504
ST		IL変数_60
LD		resBia01
AND		inBia0303
AND		IL変数_60
ST		resBia03
									
(*■CLR命令*)
(*実行されるパターン*)
LD		inCLR01
ST		resCLR01
									
LD		inCLR02
ST		resCLR02
									
(*実行されないパターン*)
LD		inCLR03
ST		resCLR03
AND		inCLR0401
AND		inCLR0402
ST		resCLR04
									
(*■DIFU(TRIGON)命令*)
LD		inDIFU
ST		R_TRIG_1.CLK
CAL		R_TRIG_1
LD		R_TRIG_1.Q
ST		outDIFU
									
LD		outDIFU
OR		holdDIFU
ST		holdDIFU
									
LDN		outDIFU
AND		holdDIFU
ST		resDIFU
									
(*■DIFD(TRIGOFF)命令*)
LD		inDIFD
ST		F_TRIG_1.CLK
CAL		F_TRIG_1
LD		F_TRIG_1.Q
ST		outDIFD
									
LD		outDIFD
OR		holdDIFD
ST		holdDIFD
									
(*-----ここまで-----------------------------------------------------
*)
LD		holdDIFD
ANDN		outDIFD
ST		resDIFD
									
								
							
						
					
						
							
								
							
							
								(*■LD命令*)
LD		input01
ST		resLD
									
(*■LDB命令*)
LDN		input01
STN		resLDB
									
(*■AND命令*)
LDN		C005
AND		input01
ST		resAND
									
(*■ANB命令*)
LDN		C007
ANDN		input01
STN		resANB
									
(*■OR命令*)
LD		C010
OR		input01
ST		resOR
									
(*■ORB命令*)
LD		C015
ORN		input01
STN		resORB
									
(*■OUT命令*)
LD		input01
ST		resOUT
									
(*■OUB命令*)
LDN		input01
STN		resOUB
									
(*■SET命令*)
LD		input01
ANDN		resSET
S		resSET
									
(*■RES命令*)
LD		input01
S		C024
									
LD		input01
R		C024
									
LDN		C024
ST		resRES
									
(*■LD_T命令*)
LD		inTIMER01
ST		TON_1.IN
ST		TON_2.IN
LD		TIME#30s
ST		TON_1.PT
CAL		TON_1
LD		TON_1.Q
ST		resTimer01
LD		TON_1.ET
ST		passed01
LD		TIME#1m
ST		TON_2.PT
CAL		TON_2
LD		TON_2.Q
ST		resTimer02
LD		TON_2.ET
ST		passed02
									
LD		resTimer01
ST		resLD_T01
									
LD		resTimer02
ST		resLD_T02
									
(*■LD_C命令*)
LD		inCounter
ST		CTU_1.CU
LD		enableCnt
ST		CTU_1.RESET
LD		INT#5000
ST		CTU_1.PV
CAL		CTU_1
LD		CTU_1.Q
ST		outConter
LD		CTU_1.CV
ST		valCounter
									
LD		outConter
ST		resLD_C
									
(*■LDB_T命令*)
LD		inTimER02
ST		TON_3.IN
LD		TIME#30s
ST		TON_3.PT
CAL		TON_3
LD		TON_3.Q
ST		resT5
LD		TON_3.ET
ST		passed03
									
LDN		resT5
STN		resLDB_T
									
(*■LDB_C命令*)
LD		inCounter2
ST		CTU_2.CU
LD		enableCnt
ST		CTU_2.RESET
LD		INT#5000
ST		CTU_2.PV
CAL		CTU_2
LD		CTU_2.Q
ST		outConter2
LD		CTU_2.CV
ST		valCounter2
									
LDN		outConter2
STN		resLDB_C
									
(*■AND_T命令*)
LD		inTimeR03
ST		TON_4.IN
LD		TIME#30s
ST		TON_4.PT
CAL		TON_4
LD		TON_4.Q
ST		outTimer
LD		TON_4.ET
ST		passed04
									
LDN		C046
AND		outTimer
ST		resAND_T
									
(*■AND_C命令*)
LD		inCounter3
ST		CTU_3.CU
LD		enableCnt
ST		CTU_3.RESET
LD		INT#5000
ST		CTU_3.PV
CAL		CTU_3
LD		CTU_3.Q
ST		outCounter3
LD		CTU_3.CV
ST		valCounter3
									
LDN		C052
AND		outCounter3
ST		resAND_C
									
(*■ANB_T命令*)
LD		inTimer05
ST		TON_5.IN
LD		TIME#30s
ST		TON_5.PT
CAL		TON_5
LD		TON_5.Q
ST		outTimer05
LD		TON_5.ET
ST		passed05
									
LDN		C055
ANDN		outTimer05
STN		resANB_T
									
(*■ANB_C命令*)
LD		inCounter04
ST		CTU_4.CU
LD		enableCnt
ST		CTU_4.RESET
LD		INT#5000
ST		CTU_4.PV
CAL		CTU_4
LD		CTU_4.Q
ST		outConter04
LD		CTU_4.CV
ST		valCounter04
									
LDN		C061
ANDN		outConter04
STN		resANB_C
									
(*■OR_T命令*)
LD		inTimer06
ST		TON_6.IN
LD		TIME#30s
ST		TON_6.PT
CAL		TON_6
LD		TON_6.Q
ST		outTimer06
LD		TON_6.ET
ST		passed06
									
LD		C065
OR		outTimer06
ST		resOR_T
									
(*■OR_C命令*)
LD		inCounter05
ST		CTU_5.CU
LD		enableCnt
ST		CTU_5.RESET
LD		INT#5000
ST		CTU_5.PV
CAL		CTU_5
LD		CTU_5.Q
ST		outCounter05
LD		CTU_5.CV
ST		valCounter05
									
LD		C069
OR		outCounter05
ST		resOR_C
									
(*■ORB_T命令*)
LD		inTimer07
ST		TON_7.IN
LD		TIME#30s
ST		TON_7.PT
CAL		TON_7
LD		TON_7.Q
ST		outTimer07
LD		TON_7.ET
ST		passed07
									
LD		C075
ORN		outTimer07
STN		resORB_T
									
(*■ORB_C命令*)
LD		inCounter06
ST		CTU_6.CU
LD		enableCnt
ST		CTU_6.RESET
LD		INT#5000
ST		CTU_6.PV
CAL		CTU_6
LD		CTU_6.Q
ST		outCounter06
LD		CTU_6.CV
ST		valCounter06
									
LD		C078
ORN		outCounter06
STN		resORB_C
									
(*■ANL命令*)
LD		input01
OR		C083
ST		IL変数_61
LD		input01
OR		C085
AND		IL変数_61
ST		resANL
									
(*■ORL命令*)
LD		input01
AND		input01
ST		IL変数_62
LD		C089
AND		C091
OR		IL変数_62
ST		resORL
									
(*■MPS、MPP、MRD命令*)
LD		setten0101
AND		setten0102
ST		IL変数_63
LD		IL変数_63
AND		setten0103
ST		IL変数_64
LD		IL変数_64
AND		setten0104
ST		resCoil01
LD		IL変数_64
AND		setten0204
ST		resCoil02
LD		IL変数_64
AND		setten0304
ST		resCoil03
LD		IL変数_63
AND		setten0403
ST		resCoil04
LD		IL変数_63
AND		setten0503
ST		resCoil05
LD		IL変数_63
AND		setten0603
ST		resCoil06
									
LD		setten0101
AND		setten0702
ST		resCoil07
									
LD		setten0101
AND		setten0802
ST		resCoil08
									
LD		setten0101
AND		setten0902
ST		resCoil09
									
(*■ビアメカ問題発生ロジック*)
LD		inBia0102
OR		inBia0202
AND		inBia0101
ST		resBia01
LD		resBia01
AND		inBia0203
ST		resBia02
LD		inBIa0404
OR		inBIa0504
ST		IL変数_65
LD		resBia01
AND		inBia0303
AND		IL変数_65
ST		resBia03
									
(*■CLR命令*)
(*実行されるパターン*)
LD		inCLR01
ST		resCLR01
									
LD		inCLR02
ST		resCLR02
									
(*実行されないパターン*)
LD		inCLR03
ST		resCLR03
AND		inCLR0401
AND		inCLR0402
ST		resCLR04
									
(*■DIFU(TRIGON)命令*)
LD		inDIFU
ST		R_TRIG_1.CLK
CAL		R_TRIG_1
LD		R_TRIG_1.Q
ST		outDIFU
									
LD		outDIFU
OR		holdDIFU
ST		holdDIFU
									
LDN		outDIFU
AND		holdDIFU
ST		resDIFU
									
(*■DIFD(TRIGOFF)命令*)
LD		inDIFD
ST		F_TRIG_1.CLK
CAL		F_TRIG_1
LD		F_TRIG_1.Q
ST		outDIFD
									
LD		outDIFD
OR		holdDIFD
ST		holdDIFD
									
(*-----ここまで-----------------------------------------------------
*)
LD		holdDIFD
ANDN		outDIFD
ST		resDIFD
									
								
							
						
					
						
							
								
							
							
								(*■LD命令*)
LD		input01
ST		resLD
									
(*■LDB命令*)
LDN		input01
STN		resLDB
									
(*■AND命令*)
LDN		C005
AND		input01
ST		resAND
									
(*■ANB命令*)
LDN		C007
ANDN		input01
STN		resANB
									
(*■OR命令*)
LD		C010
OR		input01
ST		resOR
									
(*■ORB命令*)
LD		C015
ORN		input01
STN		resORB
									
(*■OUT命令*)
LD		input01
ST		resOUT
									
(*■OUB命令*)
LDN		input01
STN		resOUB
									
(*■SET命令*)
LD		input01
ANDN		resSET
S		resSET
									
(*■RES命令*)
LD		input01
S		C024
									
LD		input01
R		C024
									
LDN		C024
ST		resRES
									
(*■LD_T命令*)
LD		inTIMER01
ST		TON_1.IN
ST		TON_2.IN
LD		TIME#30s
ST		TON_1.PT
CAL		TON_1
LD		TON_1.Q
ST		resTimer01
LD		TON_1.ET
ST		passed01
LD		TIME#1m
ST		TON_2.PT
CAL		TON_2
LD		TON_2.Q
ST		resTimer02
LD		TON_2.ET
ST		passed02
									
LD		resTimer01
ST		resLD_T01
									
LD		resTimer02
ST		resLD_T02
									
(*■LD_C命令*)
LD		inCounter
ST		CTU_1.CU
LD		enableCnt
ST		CTU_1.RESET
LD		INT#5000
ST		CTU_1.PV
CAL		CTU_1
LD		CTU_1.Q
ST		outConter
LD		CTU_1.CV
ST		valCounter
									
LD		outConter
ST		resLD_C
									
(*■LDB_T命令*)
LD		inTimER02
ST		TON_3.IN
LD		TIME#30s
ST		TON_3.PT
CAL		TON_3
LD		TON_3.Q
ST		resT5
LD		TON_3.ET
ST		passed03
									
LDN		resT5
STN		resLDB_T
									
(*■LDB_C命令*)
LD		inCounter2
ST		CTU_2.CU
LD		enableCnt
ST		CTU_2.RESET
LD		INT#5000
ST		CTU_2.PV
CAL		CTU_2
LD		CTU_2.Q
ST		outConter2
LD		CTU_2.CV
ST		valCounter2
									
LDN		outConter2
STN		resLDB_C
									
(*■AND_T命令*)
LD		inTimeR03
ST		TON_4.IN
LD		TIME#30s
ST		TON_4.PT
CAL		TON_4
LD		TON_4.Q
ST		outTimer
LD		TON_4.ET
ST		passed04
									
LDN		C046
AND		outTimer
ST		resAND_T
									
(*■AND_C命令*)
LD		inCounter3
ST		CTU_3.CU
LD		enableCnt
ST		CTU_3.RESET
LD		INT#5000
ST		CTU_3.PV
CAL		CTU_3
LD		CTU_3.Q
ST		outCounter3
LD		CTU_3.CV
ST		valCounter3
									
LDN		C052
AND		outCounter3
ST		resAND_C
									
(*■ANB_T命令*)
LD		inTimer05
ST		TON_5.IN
LD		TIME#30s
ST		TON_5.PT
CAL		TON_5
LD		TON_5.Q
ST		outTimer05
LD		TON_5.ET
ST		passed05
									
LDN		C055
ANDN		outTimer05
STN		resANB_T
									
(*■ANB_C命令*)
LD		inCounter04
ST		CTU_4.CU
LD		enableCnt
ST		CTU_4.RESET
LD		INT#5000
ST		CTU_4.PV
CAL		CTU_4
LD		CTU_4.Q
ST		outConter04
LD		CTU_4.CV
ST		valCounter04
									
LDN		C061
ANDN		outConter04
STN		resANB_C
									
(*■OR_T命令*)
LD		inTimer06
ST		TON_6.IN
LD		TIME#30s
ST		TON_6.PT
CAL		TON_6
LD		TON_6.Q
ST		outTimer06
LD		TON_6.ET
ST		passed06
									
LD		C065
OR		outTimer06
ST		resOR_T
									
(*■OR_C命令*)
LD		inCounter05
ST		CTU_5.CU
LD		enableCnt
ST		CTU_5.RESET
LD		INT#5000
ST		CTU_5.PV
CAL		CTU_5
LD		CTU_5.Q
ST		outCounter05
LD		CTU_5.CV
ST		valCounter05
									
LD		C069
OR		outCounter05
ST		resOR_C
									
(*■ORB_T命令*)
LD		inTimer07
ST		TON_7.IN
LD		TIME#30s
ST		TON_7.PT
CAL		TON_7
LD		TON_7.Q
ST		outTimer07
LD		TON_7.ET
ST		passed07
									
LD		C075
ORN		outTimer07
STN		resORB_T
									
(*■ORB_C命令*)
LD		inCounter06
ST		CTU_6.CU
LD		enableCnt
ST		CTU_6.RESET
LD		INT#5000
ST		CTU_6.PV
CAL		CTU_6
LD		CTU_6.Q
ST		outCounter06
LD		CTU_6.CV
ST		valCounter06
									
LD		C078
ORN		outCounter06
STN		resORB_C
									
(*■ANL命令*)
LD		input01
OR		C083
ST		IL変数_66
LD		input01
OR		C085
AND		IL変数_66
ST		resANL
									
(*■ORL命令*)
LD		input01
AND		input01
ST		IL変数_67
LD		C089
AND		C091
OR		IL変数_67
ST		resORL
									
(*■MPS、MPP、MRD命令*)
LD		setten0101
AND		setten0102
ST		IL変数_68
LD		IL変数_68
AND		setten0103
ST		IL変数_69
LD		IL変数_69
AND		setten0104
ST		resCoil01
LD		IL変数_69
AND		setten0204
ST		resCoil02
LD		IL変数_69
AND		setten0304
ST		resCoil03
LD		IL変数_68
AND		setten0403
ST		resCoil04
LD		IL変数_68
AND		setten0503
ST		resCoil05
LD		IL変数_68
AND		setten0603
ST		resCoil06
									
LD		setten0101
AND		setten0702
ST		resCoil07
									
LD		setten0101
AND		setten0802
ST		resCoil08
									
LD		setten0101
AND		setten0902
ST		resCoil09
									
(*■ビアメカ問題発生ロジック*)
LD		inBia0102
OR		inBia0202
AND		inBia0101
ST		resBia01
LD		resBia01
AND		inBia0203
ST		resBia02
LD		inBIa0404
OR		inBIa0504
ST		IL変数_70
LD		resBia01
AND		inBia0303
AND		IL変数_70
ST		resBia03
									
(*■CLR命令*)
(*実行されるパターン*)
LD		inCLR01
ST		resCLR01
									
LD		inCLR02
ST		resCLR02
									
(*実行されないパターン*)
LD		inCLR03
ST		resCLR03
AND		inCLR0401
AND		inCLR0402
ST		resCLR04
									
(*■DIFU(TRIGON)命令*)
LD		inDIFU
ST		R_TRIG_1.CLK
CAL		R_TRIG_1
LD		R_TRIG_1.Q
ST		outDIFU
									
LD		outDIFU
OR		holdDIFU
ST		holdDIFU
									
LDN		outDIFU
AND		holdDIFU
ST		resDIFU
									
(*■DIFD(TRIGOFF)命令*)
LD		inDIFD
ST		F_TRIG_1.CLK
CAL		F_TRIG_1
LD		F_TRIG_1.Q
ST		outDIFD
									
LD		outDIFD
OR		holdDIFD
ST		holdDIFD
									
(*-----ここまで-----------------------------------------------------
*)
LD		holdDIFD
ANDN		outDIFD
ST		resDIFD
									
								
							
						
					
						
							
								
							
							
								(*■LD命令*)
LD		input01
ST		resLD
									
(*■LDB命令*)
LDN		input01
STN		resLDB
									
(*■AND命令*)
LDN		C005
AND		input01
ST		resAND
									
(*■ANB命令*)
LDN		C007
ANDN		input01
STN		resANB
									
(*■OR命令*)
LD		C010
OR		input01
ST		resOR
									
(*■ORB命令*)
LD		C015
ORN		input01
STN		resORB
									
(*■OUT命令*)
LD		input01
ST		resOUT
									
(*■OUB命令*)
LDN		input01
STN		resOUB
									
(*■SET命令*)
LD		input01
ANDN		resSET
S		resSET
									
(*■RES命令*)
LD		input01
S		C024
									
LD		input01
R		C024
									
LDN		C024
ST		resRES
									
(*■LD_T命令*)
LD		inTIMER01
ST		TON_1.IN
ST		TON_2.IN
LD		TIME#30s
ST		TON_1.PT
CAL		TON_1
LD		TON_1.Q
ST		resTimer01
LD		TON_1.ET
ST		passed01
LD		TIME#1m
ST		TON_2.PT
CAL		TON_2
LD		TON_2.Q
ST		resTimer02
LD		TON_2.ET
ST		passed02
									
LD		resTimer01
ST		resLD_T01
									
LD		resTimer02
ST		resLD_T02
									
(*■LD_C命令*)
LD		inCounter
ST		CTU_1.CU
LD		enableCnt
ST		CTU_1.RESET
LD		INT#5000
ST		CTU_1.PV
CAL		CTU_1
LD		CTU_1.Q
ST		outConter
LD		CTU_1.CV
ST		valCounter
									
LD		outConter
ST		resLD_C
									
(*■LDB_T命令*)
LD		inTimER02
ST		TON_3.IN
LD		TIME#30s
ST		TON_3.PT
CAL		TON_3
LD		TON_3.Q
ST		resT5
LD		TON_3.ET
ST		passed03
									
LDN		resT5
STN		resLDB_T
									
(*■LDB_C命令*)
LD		inCounter2
ST		CTU_2.CU
LD		enableCnt
ST		CTU_2.RESET
LD		INT#5000
ST		CTU_2.PV
CAL		CTU_2
LD		CTU_2.Q
ST		outConter2
LD		CTU_2.CV
ST		valCounter2
									
LDN		outConter2
STN		resLDB_C
									
(*■AND_T命令*)
LD		inTimeR03
ST		TON_4.IN
LD		TIME#30s
ST		TON_4.PT
CAL		TON_4
LD		TON_4.Q
ST		outTimer
LD		TON_4.ET
ST		passed04
									
LDN		C046
AND		outTimer
ST		resAND_T
									
(*■AND_C命令*)
LD		inCounter3
ST		CTU_3.CU
LD		enableCnt
ST		CTU_3.RESET
LD		INT#5000
ST		CTU_3.PV
CAL		CTU_3
LD		CTU_3.Q
ST		outCounter3
LD		CTU_3.CV
ST		valCounter3
									
LDN		C052
AND		outCounter3
ST		resAND_C
									
(*■ANB_T命令*)
LD		inTimer05
ST		TON_5.IN
LD		TIME#30s
ST		TON_5.PT
CAL		TON_5
LD		TON_5.Q
ST		outTimer05
LD		TON_5.ET
ST		passed05
									
LDN		C055
ANDN		outTimer05
STN		resANB_T
									
(*■ANB_C命令*)
LD		inCounter04
ST		CTU_4.CU
LD		enableCnt
ST		CTU_4.RESET
LD		INT#5000
ST		CTU_4.PV
CAL		CTU_4
LD		CTU_4.Q
ST		outConter04
LD		CTU_4.CV
ST		valCounter04
									
LDN		C061
ANDN		outConter04
STN		resANB_C
									
(*■OR_T命令*)
LD		inTimer06
ST		TON_6.IN
LD		TIME#30s
ST		TON_6.PT
CAL		TON_6
LD		TON_6.Q
ST		outTimer06
LD		TON_6.ET
ST		passed06
									
LD		C065
OR		outTimer06
ST		resOR_T
									
(*■OR_C命令*)
LD		inCounter05
ST		CTU_5.CU
LD		enableCnt
ST		CTU_5.RESET
LD		INT#5000
ST		CTU_5.PV
CAL		CTU_5
LD		CTU_5.Q
ST		outCounter05
LD		CTU_5.CV
ST		valCounter05
									
LD		C069
OR		outCounter05
ST		resOR_C
									
(*■ORB_T命令*)
LD		inTimer07
ST		TON_7.IN
LD		TIME#30s
ST		TON_7.PT
CAL		TON_7
LD		TON_7.Q
ST		outTimer07
LD		TON_7.ET
ST		passed07
									
LD		C075
ORN		outTimer07
STN		resORB_T
									
(*■ORB_C命令*)
LD		inCounter06
ST		CTU_6.CU
LD		enableCnt
ST		CTU_6.RESET
LD		INT#5000
ST		CTU_6.PV
CAL		CTU_6
LD		CTU_6.Q
ST		outCounter06
LD		CTU_6.CV
ST		valCounter06
									
LD		C078
ORN		outCounter06
STN		resORB_C
									
(*■ANL命令*)
LD		input01
OR		C083
ST		IL変数_71
LD		input01
OR		C085
AND		IL変数_71
ST		resANL
									
(*■ORL命令*)
LD		input01
AND		input01
ST		IL変数_72
LD		C089
AND		C091
OR		IL変数_72
ST		resORL
									
(*■MPS、MPP、MRD命令*)
LD		setten0101
AND		setten0102
ST		IL変数_73
LD		IL変数_73
AND		setten0103
ST		IL変数_74
LD		IL変数_74
AND		setten0104
ST		resCoil01
LD		IL変数_74
AND		setten0204
ST		resCoil02
LD		IL変数_74
AND		setten0304
ST		resCoil03
LD		IL変数_73
AND		setten0403
ST		resCoil04
LD		IL変数_73
AND		setten0503
ST		resCoil05
LD		IL変数_73
AND		setten0603
ST		resCoil06
									
LD		setten0101
AND		setten0702
ST		resCoil07
									
LD		setten0101
AND		setten0802
ST		resCoil08
									
LD		setten0101
AND		setten0902
ST		resCoil09
									
(*■ビアメカ問題発生ロジック*)
LD		inBia0102
OR		inBia0202
AND		inBia0101
ST		resBia01
LD		resBia01
AND		inBia0203
ST		resBia02
LD		inBIa0404
OR		inBIa0504
ST		IL変数_75
LD		resBia01
AND		inBia0303
AND		IL変数_75
ST		resBia03
									
(*■CLR命令*)
(*実行されるパターン*)
LD		inCLR01
ST		resCLR01
									
LD		inCLR02
ST		resCLR02
									
(*実行されないパターン*)
LD		inCLR03
ST		resCLR03
AND		inCLR0401
AND		inCLR0402
ST		resCLR04
									
(*■DIFU(TRIGON)命令*)
LD		inDIFU
ST		R_TRIG_1.CLK
CAL		R_TRIG_1
LD		R_TRIG_1.Q
ST		outDIFU
									
LD		outDIFU
OR		holdDIFU
ST		holdDIFU
									
LDN		outDIFU
AND		holdDIFU
ST		resDIFU
									
(*■DIFD(TRIGOFF)命令*)
LD		inDIFD
ST		F_TRIG_1.CLK
CAL		F_TRIG_1
LD		F_TRIG_1.Q
ST		outDIFD
									
LD		outDIFD
OR		holdDIFD
ST		holdDIFD
									
(*-----ここまで-----------------------------------------------------
*)
LD		holdDIFD
ANDN		outDIFD
ST		resDIFD
									
								
							
						
					
						
							
								
							
							
								(*■LD命令*)
LD		input01
ST		resLD
									
(*■LDB命令*)
LDN		input01
STN		resLDB
									
(*■AND命令*)
LDN		C005
AND		input01
ST		resAND
									
(*■ANB命令*)
LDN		C007
ANDN		input01
STN		resANB
									
(*■OR命令*)
LD		C010
OR		input01
ST		resOR
									
(*■ORB命令*)
LD		C015
ORN		input01
STN		resORB
									
(*■OUT命令*)
LD		input01
ST		resOUT
									
(*■OUB命令*)
LDN		input01
STN		resOUB
									
(*■SET命令*)
LD		input01
ANDN		resSET
S		resSET
									
(*■RES命令*)
LD		input01
S		C024
									
LD		input01
R		C024
									
LDN		C024
ST		resRES
									
(*■LD_T命令*)
LD		inTIMER01
ST		TON_1.IN
ST		TON_2.IN
LD		TIME#30s
ST		TON_1.PT
CAL		TON_1
LD		TON_1.Q
ST		resTimer01
LD		TON_1.ET
ST		passed01
LD		TIME#1m
ST		TON_2.PT
CAL		TON_2
LD		TON_2.Q
ST		resTimer02
LD		TON_2.ET
ST		passed02
									
LD		resTimer01
ST		resLD_T01
									
LD		resTimer02
ST		resLD_T02
									
(*■LD_C命令*)
LD		inCounter
ST		CTU_1.CU
LD		enableCnt
ST		CTU_1.RESET
LD		INT#5000
ST		CTU_1.PV
CAL		CTU_1
LD		CTU_1.Q
ST		outConter
LD		CTU_1.CV
ST		valCounter
									
LD		outConter
ST		resLD_C
									
(*■LDB_T命令*)
LD		inTimER02
ST		TON_3.IN
LD		TIME#30s
ST		TON_3.PT
CAL		TON_3
LD		TON_3.Q
ST		resT5
LD		TON_3.ET
ST		passed03
									
LDN		resT5
STN		resLDB_T
									
(*■LDB_C命令*)
LD		inCounter2
ST		CTU_2.CU
LD		enableCnt
ST		CTU_2.RESET
LD		INT#5000
ST		CTU_2.PV
CAL		CTU_2
LD		CTU_2.Q
ST		outConter2
LD		CTU_2.CV
ST		valCounter2
									
LDN		outConter2
STN		resLDB_C
									
(*■AND_T命令*)
LD		inTimeR03
ST		TON_4.IN
LD		TIME#30s
ST		TON_4.PT
CAL		TON_4
LD		TON_4.Q
ST		outTimer
LD		TON_4.ET
ST		passed04
									
LDN		C046
AND		outTimer
ST		resAND_T
									
(*■AND_C命令*)
LD		inCounter3
ST		CTU_3.CU
LD		enableCnt
ST		CTU_3.RESET
LD		INT#5000
ST		CTU_3.PV
CAL		CTU_3
LD		CTU_3.Q
ST		outCounter3
LD		CTU_3.CV
ST		valCounter3
									
LDN		C052
AND		outCounter3
ST		resAND_C
									
(*■ANB_T命令*)
LD		inTimer05
ST		TON_5.IN
LD		TIME#30s
ST		TON_5.PT
CAL		TON_5
LD		TON_5.Q
ST		outTimer05
LD		TON_5.ET
ST		passed05
									
LDN		C055
ANDN		outTimer05
STN		resANB_T
									
(*■ANB_C命令*)
LD		inCounter04
ST		CTU_4.CU
LD		enableCnt
ST		CTU_4.RESET
LD		INT#5000
ST		CTU_4.PV
CAL		CTU_4
LD		CTU_4.Q
ST		outConter04
LD		CTU_4.CV
ST		valCounter04
									
LDN		C061
ANDN		outConter04
STN		resANB_C
									
(*■OR_T命令*)
LD		inTimer06
ST		TON_6.IN
LD		TIME#30s
ST		TON_6.PT
CAL		TON_6
LD		TON_6.Q
ST		outTimer06
LD		TON_6.ET
ST		passed06
									
LD		C065
OR		outTimer06
ST		resOR_T
									
(*■OR_C命令*)
LD		inCounter05
ST		CTU_5.CU
LD		enableCnt
ST		CTU_5.RESET
LD		INT#5000
ST		CTU_5.PV
CAL		CTU_5
LD		CTU_5.Q
ST		outCounter05
LD		CTU_5.CV
ST		valCounter05
									
LD		C069
OR		outCounter05
ST		resOR_C
									
(*■ORB_T命令*)
LD		inTimer07
ST		TON_7.IN
LD		TIME#30s
ST		TON_7.PT
CAL		TON_7
LD		TON_7.Q
ST		outTimer07
LD		TON_7.ET
ST		passed07
									
LD		C075
ORN		outTimer07
STN		resORB_T
									
(*■ORB_C命令*)
LD		inCounter06
ST		CTU_6.CU
LD		enableCnt
ST		CTU_6.RESET
LD		INT#5000
ST		CTU_6.PV
CAL		CTU_6
LD		CTU_6.Q
ST		outCounter06
LD		CTU_6.CV
ST		valCounter06
									
LD		C078
ORN		outCounter06
STN		resORB_C
									
(*■ANL命令*)
LD		input01
OR		C083
ST		IL変数_76
LD		input01
OR		C085
AND		IL変数_76
ST		resANL
									
(*■ORL命令*)
LD		input01
AND		input01
ST		IL変数_77
LD		C089
AND		C091
OR		IL変数_77
ST		resORL
									
(*■MPS、MPP、MRD命令*)
LD		setten0101
AND		setten0102
ST		IL変数_78
LD		IL変数_78
AND		setten0103
ST		IL変数_79
LD		IL変数_79
AND		setten0104
ST		resCoil01
LD		IL変数_79
AND		setten0204
ST		resCoil02
LD		IL変数_79
AND		setten0304
ST		resCoil03
LD		IL変数_78
AND		setten0403
ST		resCoil04
LD		IL変数_78
AND		setten0503
ST		resCoil05
LD		IL変数_78
AND		setten0603
ST		resCoil06
									
LD		setten0101
AND		setten0702
ST		resCoil07
									
LD		setten0101
AND		setten0802
ST		resCoil08
									
LD		setten0101
AND		setten0902
ST		resCoil09
									
(*■ビアメカ問題発生ロジック*)
LD		inBia0102
OR		inBia0202
AND		inBia0101
ST		resBia01
LD		resBia01
AND		inBia0203
ST		resBia02
LD		inBIa0404
OR		inBIa0504
ST		IL変数_80
LD		resBia01
AND		inBia0303
AND		IL変数_80
ST		resBia03
									
(*■CLR命令*)
(*実行されるパターン*)
LD		inCLR01
ST		resCLR01
									
LD		inCLR02
ST		resCLR02
									
(*実行されないパターン*)
LD		inCLR03
ST		resCLR03
AND		inCLR0401
AND		inCLR0402
ST		resCLR04
									
(*■DIFU(TRIGON)命令*)
LD		inDIFU
ST		R_TRIG_1.CLK
CAL		R_TRIG_1
LD		R_TRIG_1.Q
ST		outDIFU
									
LD		outDIFU
OR		holdDIFU
ST		holdDIFU
									
LDN		outDIFU
AND		holdDIFU
ST		resDIFU
									
(*■DIFD(TRIGOFF)命令*)
LD		inDIFD
ST		F_TRIG_1.CLK
CAL		F_TRIG_1
LD		F_TRIG_1.Q
ST		outDIFD
									
LD		outDIFD
OR		holdDIFD
ST		holdDIFD
									
(*-----ここまで-----------------------------------------------------
*)
LD		holdDIFD
ANDN		outDIFD
ST		resDIFD
									
								
							
						
					
						
							
								
							
							
								(*■LD命令*)
LD		input01
ST		resLD
									
(*■LDB命令*)
LDN		input01
STN		resLDB
									
(*■AND命令*)
LDN		C005
AND		input01
ST		resAND
									
(*■ANB命令*)
LDN		C007
ANDN		input01
STN		resANB
									
(*■OR命令*)
LD		C010
OR		input01
ST		resOR
									
(*■ORB命令*)
LD		C015
ORN		input01
STN		resORB
									
(*■OUT命令*)
LD		input01
ST		resOUT
									
(*■OUB命令*)
LDN		input01
STN		resOUB
									
(*■SET命令*)
LD		input01
ANDN		resSET
S		resSET
									
(*■RES命令*)
LD		input01
S		C024
									
LD		input01
R		C024
									
LDN		C024
ST		resRES
									
(*■LD_T命令*)
LD		inTIMER01
ST		TON_1.IN
ST		TON_2.IN
LD		TIME#30s
ST		TON_1.PT
CAL		TON_1
LD		TON_1.Q
ST		resTimer01
LD		TON_1.ET
ST		passed01
LD		TIME#1m
ST		TON_2.PT
CAL		TON_2
LD		TON_2.Q
ST		resTimer02
LD		TON_2.ET
ST		passed02
									
LD		resTimer01
ST		resLD_T01
									
LD		resTimer02
ST		resLD_T02
									
(*■LD_C命令*)
LD		inCounter
ST		CTU_1.CU
LD		enableCnt
ST		CTU_1.RESET
LD		INT#5000
ST		CTU_1.PV
CAL		CTU_1
LD		CTU_1.Q
ST		outConter
LD		CTU_1.CV
ST		valCounter
									
LD		outConter
ST		resLD_C
									
(*■LDB_T命令*)
LD		inTimER02
ST		TON_3.IN
LD		TIME#30s
ST		TON_3.PT
CAL		TON_3
LD		TON_3.Q
ST		resT5
LD		TON_3.ET
ST		passed03
									
LDN		resT5
STN		resLDB_T
									
(*■LDB_C命令*)
LD		inCounter2
ST		CTU_2.CU
LD		enableCnt
ST		CTU_2.RESET
LD		INT#5000
ST		CTU_2.PV
CAL		CTU_2
LD		CTU_2.Q
ST		outConter2
LD		CTU_2.CV
ST		valCounter2
									
LDN		outConter2
STN		resLDB_C
									
(*■AND_T命令*)
LD		inTimeR03
ST		TON_4.IN
LD		TIME#30s
ST		TON_4.PT
CAL		TON_4
LD		TON_4.Q
ST		outTimer
LD		TON_4.ET
ST		passed04
									
LDN		C046
AND		outTimer
ST		resAND_T
									
(*■AND_C命令*)
LD		inCounter3
ST		CTU_3.CU
LD		enableCnt
ST		CTU_3.RESET
LD		INT#5000
ST		CTU_3.PV
CAL		CTU_3
LD		CTU_3.Q
ST		outCounter3
LD		CTU_3.CV
ST		valCounter3
									
LDN		C052
AND		outCounter3
ST		resAND_C
									
(*■ANB_T命令*)
LD		inTimer05
ST		TON_5.IN
LD		TIME#30s
ST		TON_5.PT
CAL		TON_5
LD		TON_5.Q
ST		outTimer05
LD		TON_5.ET
ST		passed05
									
LDN		C055
ANDN		outTimer05
STN		resANB_T
									
(*■ANB_C命令*)
LD		inCounter04
ST		CTU_4.CU
LD		enableCnt
ST		CTU_4.RESET
LD		INT#5000
ST		CTU_4.PV
CAL		CTU_4
LD		CTU_4.Q
ST		outConter04
LD		CTU_4.CV
ST		valCounter04
									
LDN		C061
ANDN		outConter04
STN		resANB_C
									
(*■OR_T命令*)
LD		inTimer06
ST		TON_6.IN
LD		TIME#30s
ST		TON_6.PT
CAL		TON_6
LD		TON_6.Q
ST		outTimer06
LD		TON_6.ET
ST		passed06
									
LD		C065
OR		outTimer06
ST		resOR_T
									
(*■OR_C命令*)
LD		inCounter05
ST		CTU_5.CU
LD		enableCnt
ST		CTU_5.RESET
LD		INT#5000
ST		CTU_5.PV
CAL		CTU_5
LD		CTU_5.Q
ST		outCounter05
LD		CTU_5.CV
ST		valCounter05
									
LD		C069
OR		outCounter05
ST		resOR_C
									
(*■ORB_T命令*)
LD		inTimer07
ST		TON_7.IN
LD		TIME#30s
ST		TON_7.PT
CAL		TON_7
LD		TON_7.Q
ST		outTimer07
LD		TON_7.ET
ST		passed07
									
LD		C075
ORN		outTimer07
STN		resORB_T
									
(*■ORB_C命令*)
LD		inCounter06
ST		CTU_6.CU
LD		enableCnt
ST		CTU_6.RESET
LD		INT#5000
ST		CTU_6.PV
CAL		CTU_6
LD		CTU_6.Q
ST		outCounter06
LD		CTU_6.CV
ST		valCounter06
									
LD		C078
ORN		outCounter06
STN		resORB_C
									
(*■ANL命令*)
LD		input01
OR		C083
ST		IL変数_81
LD		input01
OR		C085
AND		IL変数_81
ST		resANL
									
(*■ORL命令*)
LD		input01
AND		input01
ST		IL変数_82
LD		C089
AND		C091
OR		IL変数_82
ST		resORL
									
(*■MPS、MPP、MRD命令*)
LD		setten0101
AND		setten0102
ST		IL変数_83
LD		IL変数_83
AND		setten0103
ST		IL変数_84
LD		IL変数_84
AND		setten0104
ST		resCoil01
LD		IL変数_84
AND		setten0204
ST		resCoil02
LD		IL変数_84
AND		setten0304
ST		resCoil03
LD		IL変数_83
AND		setten0403
ST		resCoil04
LD		IL変数_83
AND		setten0503
ST		resCoil05
LD		IL変数_83
AND		setten0603
ST		resCoil06
									
LD		setten0101
AND		setten0702
ST		resCoil07
									
LD		setten0101
AND		setten0802
ST		resCoil08
									
LD		setten0101
AND		setten0902
ST		resCoil09
									
(*■ビアメカ問題発生ロジック*)
LD		inBia0102
OR		inBia0202
AND		inBia0101
ST		resBia01
LD		resBia01
AND		inBia0203
ST		resBia02
LD		inBIa0404
OR		inBIa0504
ST		IL変数_85
LD		resBia01
AND		inBia0303
AND		IL変数_85
ST		resBia03
									
(*■CLR命令*)
(*実行されるパターン*)
LD		inCLR01
ST		resCLR01
									
LD		inCLR02
ST		resCLR02
									
(*実行されないパターン*)
LD		inCLR03
ST		resCLR03
AND		inCLR0401
AND		inCLR0402
ST		resCLR04
									
(*■DIFU(TRIGON)命令*)
LD		inDIFU
ST		R_TRIG_1.CLK
CAL		R_TRIG_1
LD		R_TRIG_1.Q
ST		outDIFU
									
LD		outDIFU
OR		holdDIFU
ST		holdDIFU
									
LDN		outDIFU
AND		holdDIFU
ST		resDIFU
									
(*■DIFD(TRIGOFF)命令*)
LD		inDIFD
ST		F_TRIG_1.CLK
CAL		F_TRIG_1
LD		F_TRIG_1.Q
ST		outDIFD
									
LD		outDIFD
OR		holdDIFD
ST		holdDIFD
									
(*-----ここまで-----------------------------------------------------
*)
LD		holdDIFD
ANDN		outDIFD
ST		resDIFD
									
								
							
						
					
						
							
								
							
							
								(*■LD命令*)
LD		input01
ST		resLD
									
(*■LDB命令*)
LDN		input01
STN		resLDB
									
(*■AND命令*)
LDN		C005
AND		input01
ST		resAND
									
(*■ANB命令*)
LDN		C007
ANDN		input01
STN		resANB
									
(*■OR命令*)
LD		C010
OR		input01
ST		resOR
									
(*■ORB命令*)
LD		C015
ORN		input01
STN		resORB
									
(*■OUT命令*)
LD		input01
ST		resOUT
									
(*■OUB命令*)
LDN		input01
STN		resOUB
									
(*■SET命令*)
LD		input01
ANDN		resSET
S		resSET
									
(*■RES命令*)
LD		input01
S		C024
									
LD		input01
R		C024
									
LDN		C024
ST		resRES
									
(*■LD_T命令*)
LD		inTIMER01
ST		TON_1.IN
ST		TON_2.IN
LD		TIME#30s
ST		TON_1.PT
CAL		TON_1
LD		TON_1.Q
ST		resTimer01
LD		TON_1.ET
ST		passed01
LD		TIME#1m
ST		TON_2.PT
CAL		TON_2
LD		TON_2.Q
ST		resTimer02
LD		TON_2.ET
ST		passed02
									
LD		resTimer01
ST		resLD_T01
									
LD		resTimer02
ST		resLD_T02
									
(*■LD_C命令*)
LD		inCounter
ST		CTU_1.CU
LD		enableCnt
ST		CTU_1.RESET
LD		INT#5000
ST		CTU_1.PV
CAL		CTU_1
LD		CTU_1.Q
ST		outConter
LD		CTU_1.CV
ST		valCounter
									
LD		outConter
ST		resLD_C
									
(*■LDB_T命令*)
LD		inTimER02
ST		TON_3.IN
LD		TIME#30s
ST		TON_3.PT
CAL		TON_3
LD		TON_3.Q
ST		resT5
LD		TON_3.ET
ST		passed03
									
LDN		resT5
STN		resLDB_T
									
(*■LDB_C命令*)
LD		inCounter2
ST		CTU_2.CU
LD		enableCnt
ST		CTU_2.RESET
LD		INT#5000
ST		CTU_2.PV
CAL		CTU_2
LD		CTU_2.Q
ST		outConter2
LD		CTU_2.CV
ST		valCounter2
									
LDN		outConter2
STN		resLDB_C
									
(*■AND_T命令*)
LD		inTimeR03
ST		TON_4.IN
LD		TIME#30s
ST		TON_4.PT
CAL		TON_4
LD		TON_4.Q
ST		outTimer
LD		TON_4.ET
ST		passed04
									
LDN		C046
AND		outTimer
ST		resAND_T
									
(*■AND_C命令*)
LD		inCounter3
ST		CTU_3.CU
LD		enableCnt
ST		CTU_3.RESET
LD		INT#5000
ST		CTU_3.PV
CAL		CTU_3
LD		CTU_3.Q
ST		outCounter3
LD		CTU_3.CV
ST		valCounter3
									
LDN		C052
AND		outCounter3
ST		resAND_C
									
(*■ANB_T命令*)
LD		inTimer05
ST		TON_5.IN
LD		TIME#30s
ST		TON_5.PT
CAL		TON_5
LD		TON_5.Q
ST		outTimer05
LD		TON_5.ET
ST		passed05
									
LDN		C055
ANDN		outTimer05
STN		resANB_T
									
(*■ANB_C命令*)
LD		inCounter04
ST		CTU_4.CU
LD		enableCnt
ST		CTU_4.RESET
LD		INT#5000
ST		CTU_4.PV
CAL		CTU_4
LD		CTU_4.Q
ST		outConter04
LD		CTU_4.CV
ST		valCounter04
									
LDN		C061
ANDN		outConter04
STN		resANB_C
									
(*■OR_T命令*)
LD		inTimer06
ST		TON_6.IN
LD		TIME#30s
ST		TON_6.PT
CAL		TON_6
LD		TON_6.Q
ST		outTimer06
LD		TON_6.ET
ST		passed06
									
LD		C065
OR		outTimer06
ST		resOR_T
									
(*■OR_C命令*)
LD		inCounter05
ST		CTU_5.CU
LD		enableCnt
ST		CTU_5.RESET
LD		INT#5000
ST		CTU_5.PV
CAL		CTU_5
LD		CTU_5.Q
ST		outCounter05
LD		CTU_5.CV
ST		valCounter05
									
LD		C069
OR		outCounter05
ST		resOR_C
									
(*■ORB_T命令*)
LD		inTimer07
ST		TON_7.IN
LD		TIME#30s
ST		TON_7.PT
CAL		TON_7
LD		TON_7.Q
ST		outTimer07
LD		TON_7.ET
ST		passed07
									
LD		C075
ORN		outTimer07
STN		resORB_T
									
(*■ORB_C命令*)
LD		inCounter06
ST		CTU_6.CU
LD		enableCnt
ST		CTU_6.RESET
LD		INT#5000
ST		CTU_6.PV
CAL		CTU_6
LD		CTU_6.Q
ST		outCounter06
LD		CTU_6.CV
ST		valCounter06
									
LD		C078
ORN		outCounter06
STN		resORB_C
									
(*■ANL命令*)
LD		input01
OR		C083
ST		IL変数_86
LD		input01
OR		C085
AND		IL変数_86
ST		resANL
									
(*■ORL命令*)
LD		input01
AND		input01
ST		IL変数_87
LD		C089
AND		C091
OR		IL変数_87
ST		resORL
									
(*■MPS、MPP、MRD命令*)
LD		setten0101
AND		setten0102
ST		IL変数_88
LD		IL変数_88
AND		setten0103
ST		IL変数_89
LD		IL変数_89
AND		setten0104
ST		resCoil01
LD		IL変数_89
AND		setten0204
ST		resCoil02
LD		IL変数_89
AND		setten0304
ST		resCoil03
LD		IL変数_88
AND		setten0403
ST		resCoil04
LD		IL変数_88
AND		setten0503
ST		resCoil05
LD		IL変数_88
AND		setten0603
ST		resCoil06
									
LD		setten0101
AND		setten0702
ST		resCoil07
									
LD		setten0101
AND		setten0802
ST		resCoil08
									
LD		setten0101
AND		setten0902
ST		resCoil09
									
(*■ビアメカ問題発生ロジック*)
LD		inBia0102
OR		inBia0202
AND		inBia0101
ST		resBia01
LD		resBia01
AND		inBia0203
ST		resBia02
LD		inBIa0404
OR		inBIa0504
ST		IL変数_90
LD		resBia01
AND		inBia0303
AND		IL変数_90
ST		resBia03
									
(*■CLR命令*)
(*実行されるパターン*)
LD		inCLR01
ST		resCLR01
									
LD		inCLR02
ST		resCLR02
									
(*実行されないパターン*)
LD		inCLR03
ST		resCLR03
AND		inCLR0401
AND		inCLR0402
ST		resCLR04
									
(*■DIFU(TRIGON)命令*)
LD		inDIFU
ST		R_TRIG_1.CLK
CAL		R_TRIG_1
LD		R_TRIG_1.Q
ST		outDIFU
									
LD		outDIFU
OR		holdDIFU
ST		holdDIFU
									
LDN		outDIFU
AND		holdDIFU
ST		resDIFU
									
(*■DIFD(TRIGOFF)命令*)
LD		inDIFD
ST		F_TRIG_1.CLK
CAL		F_TRIG_1
LD		F_TRIG_1.Q
ST		outDIFD
									
LD		outDIFD
OR		holdDIFD
ST		holdDIFD
									
(*-----ここまで-----------------------------------------------------
*)
LD		holdDIFD
ANDN		outDIFD
ST		resDIFD
									
								
							
						
					
						
							
								
							
							
								(*■LD命令*)
LD		input01
ST		resLD
									
(*■LDB命令*)
LDN		input01
STN		resLDB
									
(*■AND命令*)
LDN		C005
AND		input01
ST		resAND
									
(*■ANB命令*)
LDN		C007
ANDN		input01
STN		resANB
									
(*■OR命令*)
LD		C010
OR		input01
ST		resOR
									
(*■ORB命令*)
LD		C015
ORN		input01
STN		resORB
									
(*■OUT命令*)
LD		input01
ST		resOUT
									
(*■OUB命令*)
LDN		input01
STN		resOUB
									
(*■SET命令*)
LD		input01
ANDN		resSET
S		resSET
									
(*■RES命令*)
LD		input01
S		C024
									
LD		input01
R		C024
									
LDN		C024
ST		resRES
									
(*■LD_T命令*)
LD		inTIMER01
ST		TON_1.IN
ST		TON_2.IN
LD		TIME#30s
ST		TON_1.PT
CAL		TON_1
LD		TON_1.Q
ST		resTimer01
LD		TON_1.ET
ST		passed01
LD		TIME#1m
ST		TON_2.PT
CAL		TON_2
LD		TON_2.Q
ST		resTimer02
LD		TON_2.ET
ST		passed02
									
LD		resTimer01
ST		resLD_T01
									
LD		resTimer02
ST		resLD_T02
									
(*■LD_C命令*)
LD		inCounter
ST		CTU_1.CU
LD		enableCnt
ST		CTU_1.RESET
LD		INT#5000
ST		CTU_1.PV
CAL		CTU_1
LD		CTU_1.Q
ST		outConter
LD		CTU_1.CV
ST		valCounter
									
LD		outConter
ST		resLD_C
									
(*■LDB_T命令*)
LD		inTimER02
ST		TON_3.IN
LD		TIME#30s
ST		TON_3.PT
CAL		TON_3
LD		TON_3.Q
ST		resT5
LD		TON_3.ET
ST		passed03
									
LDN		resT5
STN		resLDB_T
									
(*■LDB_C命令*)
LD		inCounter2
ST		CTU_2.CU
LD		enableCnt
ST		CTU_2.RESET
LD		INT#5000
ST		CTU_2.PV
CAL		CTU_2
LD		CTU_2.Q
ST		outConter2
LD		CTU_2.CV
ST		valCounter2
									
LDN		outConter2
STN		resLDB_C
									
(*■AND_T命令*)
LD		inTimeR03
ST		TON_4.IN
LD		TIME#30s
ST		TON_4.PT
CAL		TON_4
LD		TON_4.Q
ST		outTimer
LD		TON_4.ET
ST		passed04
									
LDN		C046
AND		outTimer
ST		resAND_T
									
(*■AND_C命令*)
LD		inCounter3
ST		CTU_3.CU
LD		enableCnt
ST		CTU_3.RESET
LD		INT#5000
ST		CTU_3.PV
CAL		CTU_3
LD		CTU_3.Q
ST		outCounter3
LD		CTU_3.CV
ST		valCounter3
									
LDN		C052
AND		outCounter3
ST		resAND_C
									
(*■ANB_T命令*)
LD		inTimer05
ST		TON_5.IN
LD		TIME#30s
ST		TON_5.PT
CAL		TON_5
LD		TON_5.Q
ST		outTimer05
LD		TON_5.ET
ST		passed05
									
LDN		C055
ANDN		outTimer05
STN		resANB_T
									
(*■ANB_C命令*)
LD		inCounter04
ST		CTU_4.CU
LD		enableCnt
ST		CTU_4.RESET
LD		INT#5000
ST		CTU_4.PV
CAL		CTU_4
LD		CTU_4.Q
ST		outConter04
LD		CTU_4.CV
ST		valCounter04
									
LDN		C061
ANDN		outConter04
STN		resANB_C
									
(*■OR_T命令*)
LD		inTimer06
ST		TON_6.IN
LD		TIME#30s
ST		TON_6.PT
CAL		TON_6
LD		TON_6.Q
ST		outTimer06
LD		TON_6.ET
ST		passed06
									
LD		C065
OR		outTimer06
ST		resOR_T
									
(*■OR_C命令*)
LD		inCounter05
ST		CTU_5.CU
LD		enableCnt
ST		CTU_5.RESET
LD		INT#5000
ST		CTU_5.PV
CAL		CTU_5
LD		CTU_5.Q
ST		outCounter05
LD		CTU_5.CV
ST		valCounter05
									
LD		C069
OR		outCounter05
ST		resOR_C
									
(*■ORB_T命令*)
LD		inTimer07
ST		TON_7.IN
LD		TIME#30s
ST		TON_7.PT
CAL		TON_7
LD		TON_7.Q
ST		outTimer07
LD		TON_7.ET
ST		passed07
									
LD		C075
ORN		outTimer07
STN		resORB_T
									
(*■ORB_C命令*)
LD		inCounter06
ST		CTU_6.CU
LD		enableCnt
ST		CTU_6.RESET
LD		INT#5000
ST		CTU_6.PV
CAL		CTU_6
LD		CTU_6.Q
ST		outCounter06
LD		CTU_6.CV
ST		valCounter06
									
LD		C078
ORN		outCounter06
STN		resORB_C
									
(*■ANL命令*)
LD		input01
OR		C083
ST		IL変数_91
LD		input01
OR		C085
AND		IL変数_91
ST		resANL
									
(*■ORL命令*)
LD		input01
AND		input01
ST		IL変数_92
LD		C089
AND		C091
OR		IL変数_92
ST		resORL
									
(*■MPS、MPP、MRD命令*)
LD		setten0101
AND		setten0102
ST		IL変数_93
LD		IL変数_93
AND		setten0103
ST		IL変数_94
LD		IL変数_94
AND		setten0104
ST		resCoil01
LD		IL変数_94
AND		setten0204
ST		resCoil02
LD		IL変数_94
AND		setten0304
ST		resCoil03
LD		IL変数_93
AND		setten0403
ST		resCoil04
LD		IL変数_93
AND		setten0503
ST		resCoil05
LD		IL変数_93
AND		setten0603
ST		resCoil06
									
LD		setten0101
AND		setten0702
ST		resCoil07
									
LD		setten0101
AND		setten0802
ST		resCoil08
									
LD		setten0101
AND		setten0902
ST		resCoil09
									
(*■ビアメカ問題発生ロジック*)
LD		inBia0102
OR		inBia0202
AND		inBia0101
ST		resBia01
LD		resBia01
AND		inBia0203
ST		resBia02
LD		inBIa0404
OR		inBIa0504
ST		IL変数_95
LD		resBia01
AND		inBia0303
AND		IL変数_95
ST		resBia03
									
(*■CLR命令*)
(*実行されるパターン*)
LD		inCLR01
ST		resCLR01
									
LD		inCLR02
ST		resCLR02
									
(*実行されないパターン*)
LD		inCLR03
ST		resCLR03
AND		inCLR0401
AND		inCLR0402
ST		resCLR04
									
(*■DIFU(TRIGON)命令*)
LD		inDIFU
ST		R_TRIG_1.CLK
CAL		R_TRIG_1
LD		R_TRIG_1.Q
ST		outDIFU
									
LD		outDIFU
OR		holdDIFU
ST		holdDIFU
									
LDN		outDIFU
AND		holdDIFU
ST		resDIFU
									
(*■DIFD(TRIGOFF)命令*)
LD		inDIFD
ST		F_TRIG_1.CLK
CAL		F_TRIG_1
LD		F_TRIG_1.Q
ST		outDIFD
									
LD		outDIFD
OR		holdDIFD
ST		holdDIFD
									
(*-----ここまで-----------------------------------------------------
*)
LD		holdDIFD
ANDN		outDIFD
ST		resDIFD
									
								
							
						
					
						
							
								
							
							
								(*■LD命令*)
LD		input01
ST		resLD
									
(*■LDB命令*)
LDN		input01
STN		resLDB
									
(*■AND命令*)
LDN		C005
AND		input01
ST		resAND
									
(*■ANB命令*)
LDN		C007
ANDN		input01
STN		resANB
									
(*■OR命令*)
LD		C010
OR		input01
ST		resOR
									
(*■ORB命令*)
LD		C015
ORN		input01
STN		resORB
									
(*■OUT命令*)
LD		input01
ST		resOUT
									
(*■OUB命令*)
LDN		input01
STN		resOUB
									
(*■SET命令*)
LD		input01
ANDN		resSET
S		resSET
									
(*■RES命令*)
LD		input01
S		C024
									
LD		input01
R		C024
									
LDN		C024
ST		resRES
									
(*■LD_T命令*)
LD		inTIMER01
ST		TON_1.IN
ST		TON_2.IN
LD		TIME#30s
ST		TON_1.PT
CAL		TON_1
LD		TON_1.Q
ST		resTimer01
LD		TON_1.ET
ST		passed01
LD		TIME#1m
ST		TON_2.PT
CAL		TON_2
LD		TON_2.Q
ST		resTimer02
LD		TON_2.ET
ST		passed02
									
LD		resTimer01
ST		resLD_T01
									
LD		resTimer02
ST		resLD_T02
									
(*■LD_C命令*)
LD		inCounter
ST		CTU_1.CU
LD		enableCnt
ST		CTU_1.RESET
LD		INT#5000
ST		CTU_1.PV
CAL		CTU_1
LD		CTU_1.Q
ST		outConter
LD		CTU_1.CV
ST		valCounter
									
LD		outConter
ST		resLD_C
									
(*■LDB_T命令*)
LD		inTimER02
ST		TON_3.IN
LD		TIME#30s
ST		TON_3.PT
CAL		TON_3
LD		TON_3.Q
ST		resT5
LD		TON_3.ET
ST		passed03
									
LDN		resT5
STN		resLDB_T
									
(*■LDB_C命令*)
LD		inCounter2
ST		CTU_2.CU
LD		enableCnt
ST		CTU_2.RESET
LD		INT#5000
ST		CTU_2.PV
CAL		CTU_2
LD		CTU_2.Q
ST		outConter2
LD		CTU_2.CV
ST		valCounter2
									
LDN		outConter2
STN		resLDB_C
									
(*■AND_T命令*)
LD		inTimeR03
ST		TON_4.IN
LD		TIME#30s
ST		TON_4.PT
CAL		TON_4
LD		TON_4.Q
ST		outTimer
LD		TON_4.ET
ST		passed04
									
LDN		C046
AND		outTimer
ST		resAND_T
									
(*■AND_C命令*)
LD		inCounter3
ST		CTU_3.CU
LD		enableCnt
ST		CTU_3.RESET
LD		INT#5000
ST		CTU_3.PV
CAL		CTU_3
LD		CTU_3.Q
ST		outCounter3
LD		CTU_3.CV
ST		valCounter3
									
LDN		C052
AND		outCounter3
ST		resAND_C
									
(*■ANB_T命令*)
LD		inTimer05
ST		TON_5.IN
LD		TIME#30s
ST		TON_5.PT
CAL		TON_5
LD		TON_5.Q
ST		outTimer05
LD		TON_5.ET
ST		passed05
									
LDN		C055
ANDN		outTimer05
STN		resANB_T
									
(*■ANB_C命令*)
LD		inCounter04
ST		CTU_4.CU
LD		enableCnt
ST		CTU_4.RESET
LD		INT#5000
ST		CTU_4.PV
CAL		CTU_4
LD		CTU_4.Q
ST		outConter04
LD		CTU_4.CV
ST		valCounter04
									
LDN		C061
ANDN		outConter04
STN		resANB_C
									
(*■OR_T命令*)
LD		inTimer06
ST		TON_6.IN
LD		TIME#30s
ST		TON_6.PT
CAL		TON_6
LD		TON_6.Q
ST		outTimer06
LD		TON_6.ET
ST		passed06
									
LD		C065
OR		outTimer06
ST		resOR_T
									
(*■OR_C命令*)
LD		inCounter05
ST		CTU_5.CU
LD		enableCnt
ST		CTU_5.RESET
LD		INT#5000
ST		CTU_5.PV
CAL		CTU_5
LD		CTU_5.Q
ST		outCounter05
LD		CTU_5.CV
ST		valCounter05
									
LD		C069
OR		outCounter05
ST		resOR_C
									
(*■ORB_T命令*)
LD		inTimer07
ST		TON_7.IN
LD		TIME#30s
ST		TON_7.PT
CAL		TON_7
LD		TON_7.Q
ST		outTimer07
LD		TON_7.ET
ST		passed07
									
LD		C075
ORN		outTimer07
STN		resORB_T
									
(*■ORB_C命令*)
LD		inCounter06
ST		CTU_6.CU
LD		enableCnt
ST		CTU_6.RESET
LD		INT#5000
ST		CTU_6.PV
CAL		CTU_6
LD		CTU_6.Q
ST		outCounter06
LD		CTU_6.CV
ST		valCounter06
									
LD		C078
ORN		outCounter06
STN		resORB_C
									
(*■ANL命令*)
LD		input01
OR		C083
ST		IL変数_96
LD		input01
OR		C085
AND		IL変数_96
ST		resANL
									
(*■ORL命令*)
LD		input01
AND		input01
ST		IL変数_97
LD		C089
AND		C091
OR		IL変数_97
ST		resORL
									
(*■MPS、MPP、MRD命令*)
LD		setten0101
AND		setten0102
ST		IL変数_98
LD		IL変数_98
AND		setten0103
ST		IL変数_99
LD		IL変数_99
AND		setten0104
ST		resCoil01
LD		IL変数_99
AND		setten0204
ST		resCoil02
LD		IL変数_99
AND		setten0304
ST		resCoil03
LD		IL変数_98
AND		setten0403
ST		resCoil04
LD		IL変数_98
AND		setten0503
ST		resCoil05
LD		IL変数_98
AND		setten0603
ST		resCoil06
									
LD		setten0101
AND		setten0702
ST		resCoil07
									
LD		setten0101
AND		setten0802
ST		resCoil08
									
LD		setten0101
AND		setten0902
ST		resCoil09
									
(*■ビアメカ問題発生ロジック*)
LD		inBia0102
OR		inBia0202
AND		inBia0101
ST		resBia01
LD		resBia01
AND		inBia0203
ST		resBia02
LD		inBIa0404
OR		inBIa0504
ST		IL変数_100
LD		resBia01
AND		inBia0303
AND		IL変数_100
ST		resBia03
									
(*■CLR命令*)
(*実行されるパターン*)
LD		inCLR01
ST		resCLR01
									
LD		inCLR02
ST		resCLR02
									
(*実行されないパターン*)
LD		inCLR03
ST		resCLR03
AND		inCLR0401
AND		inCLR0402
ST		resCLR04
									
(*■DIFU(TRIGON)命令*)
LD		inDIFU
ST		R_TRIG_1.CLK
CAL		R_TRIG_1
LD		R_TRIG_1.Q
ST		outDIFU
									
LD		outDIFU
OR		holdDIFU
ST		holdDIFU
									
LDN		outDIFU
AND		holdDIFU
ST		resDIFU
									
(*■DIFD(TRIGOFF)命令*)
LD		inDIFD
ST		F_TRIG_1.CLK
CAL		F_TRIG_1
LD		F_TRIG_1.Q
ST		outDIFD
									
LD		outDIFD
OR		holdDIFD
ST		holdDIFD
									
(*-----ここまで-----------------------------------------------------
*)
LD		holdDIFD
ANDN		outDIFD
ST		resDIFD
									
								
							
						
					
						
							
								
							
							
